LIN {X 0,Y 194.629,Z 450.063,A -85,B 0,C 180,E1 -23083.872,E2 -23083.872} C_VEL
LIN {X 0,Y 195.031,Z 466.842,A -85,B 0,C 180,E1 -23086.302,E2 -23086.302} C_VEL
LIN {X 0,Y 195.009,Z 478.19,A -85,B 0,C 180,E1 -23088.193,E2 -23088.193} C_VEL
LIN {X 0,Y 190.947,Z 492.409,A -85,B 0,C 180,E1 -23090.684,E2 -23090.684} C_VEL
LIN {X 0,Y 187.15,Z 505.053,A -85,B 0,C 180,E1 -23093.413,E2 -23093.413} C_VEL
LIN {X 0,Y 184.446,Z 513.327,A -85,B 0,C 180,E1 -23095.481,E2 -23095.481} C_VEL
LIN {X 0,Y 181.735,Z 524.579,A -85,B 0,C 180,E1 -23097.846,E2 -23097.846} C_VEL
LIN {X 0,Y 179.023,Z 534.861,A -85,B 0,C 180,E1 -23100.619,E2 -23100.619} C_VEL
LIN {X 0,Y 176.653,Z 543.209,A -85,B 0,C 180,E1 -23103.419,E2 -23103.419} C_VEL
LIN {X 0,Y 174.413,Z 551.586,A -85,B 0,C 180,E1 -23106.936,E2 -23106.936} C_VEL
LIN {X 0,Y 173.108,Z 557.098,A -85,B 0,C 180,E1 -23109.819,E2 -23109.819} C_VEL
LIN {X 0,Y 171.926,Z 562.635,A -85,B 0,C 180,E1 -23113.379,E2 -23113.379} C_VEL
LIN {X 0,Y 171.267,Z 566.965,A -85,B 0,C 180,E1 -23116.962,E2 -23116.962} C_VEL
LIN {X 0,Y 171.183,Z 568.089,A -85,B 0,C 180,E1 -23118.106,E2 -23118.106} C_VEL
LIN {X 0,Y 170.832,Z 569.219,A -85,B 0,C 180,E1 -23119.364,E2 -23119.364} C_VEL
LIN {X 0,Y 169.495,Z 570.537,A -85,B 0,C 180,E1 -23121.258,E2 -23121.258} C_VEL
LIN {X 0,Y 165.486,Z 572.266,A -85,B 0,C 180,E1 -23125.813,E2 -23125.813} C_VEL
LIN {X 0,Y 164.692,Z 572.641,A -85,B 0,C 180,E1 -23127.873,E2 -23127.873} C_VEL
LIN {X 0,Y 164.706,Z 572.679,A -85,B 0,C 180,E1 -23128.568,E2 -23128.568} C_VEL
LIN {X 0,Y 164.962,Z 572.852,A -85,B 0,C 180,E1 -23130.006,E2 -23130.006} C_VEL
LIN {X 0,Y 164.703,Z 572.564,A -85,B 0,C 180,E1 -23132.451,E2 -23132.451} C_VEL
LIN {X 0,Y 164.155,Z 571.139,A -85,B 0,C 180,E1 -23137.385,E2 -23137.385} C_VEL
LIN {X 0,Y 163.743,Z 570.715,A -85,B 0,C 180,E1 -23142.398,E2 -23142.398} C_VEL
LIN {X 0,Y 164.326,Z 569.479,A -85,B 0,C 180,E1 -23147.426,E2 -23147.426} C_VEL
LIN {X 0,Y 167.378,Z 566.15,A -85,B 0,C 180,E1 -23154.833,E2 -23154.833} C_VEL
LIN {X 0,Y 173.216,Z 561.282,A -85,B 0,C 180,E1 -23161.84,E2 -23161.84} C_VEL
LIN {X 0,Y 181.825,Z 555.041,A -85,B 0,C 180,E1 -23168.208,E2 -23168.208} C_VEL
LIN {X 0,Y 192.905,Z 547.519,A -85,B 0,C 180,E1 -23173.811,E2 -23173.811} C_VEL
LIN {X 0,Y 203.834,Z 540.338,A -85,B 0,C 180,E1 -23177.848,E2 -23177.848} C_VEL
LIN {X 0,Y 210.94,Z 535.655,A -85,B 0,C 180,E1 -23180.029,E2 -23180.029} C_VEL
LIN {X 0,Y 218.242,Z 530.911,A -85,B 0,C 180,E1 -23181.835,E2 -23181.835} C_VEL
LIN {X 0,Y 219.723,Z 529.675,A -85,B 0,C 180,E1 -23182.575,E2 -23182.575} C_VEL
LIN {X 0,Y 210.166,Z 532.82,A -85,B 0,C 180,E1 -23185.356,E2 -23185.356} C_VEL
LIN {X 0,Y 201.392,Z 535.122,A -85,B 0,C 180,E1 -23188.437,E2 -23188.437} C_VEL
LIN {X 0,Y 193.436,Z 536.513,A -85,B 0,C 180,E1 -23191.816,E2 -23191.816} C_VEL
LIN {X 0,Y 186.362,Z 536.937,A -85,B 0,C 180,E1 -23195.492,E2 -23195.492} C_VEL
LIN {X 0,Y 179.439,Z 536.136,A -85,B 0,C 180,E1 -23200.063,E2 -23200.063} C_VEL
LIN {X 0,Y 175.186,Z 534.57,A -85,B 0,C 180,E1 -23203.692,E2 -23203.692} C_VEL
LIN {X 0,Y 171.279,Z 531.629,A -85,B 0,C 180,E1 -23208.162,E2 -23208.162} C_VEL
LIN {X 0,Y 168.34,Z 527.424,A -85,B 0,C 180,E1 -23212.806,E2 -23212.806} C_VEL
LIN {X 0,Y 166.311,Z 521.843,A -85,B 0,C 180,E1 -23217.579,E2 -23217.579} C_VEL
LIN {X 0,Y 165.364,Z 514.747,A -85,B 0,C 180,E1 -23222.437,E2 -23222.437} C_VEL
LIN {X 0,Y 165.269,Z 507.081,A -85,B 0,C 180,E1 -23226.717,E2 -23226.717} C_VEL
LIN {X 0,Y 165.94,Z 497.974,A -85,B 0,C 180,E1 -23230.988,E2 -23230.988} C_VEL
LIN {X 0,Y 167.032,Z 488.726,A -85,B 0,C 180,E1 -23234.624,E2 -23234.624} C_VEL
LIN {X 0,Y 168.903,Z 476.078,A -85,B 0,C 180,E1 -23238.814,E2 -23238.814} C_VEL
LIN {X 0,Y 170.944,Z 463.074,A -85,B 0,C 180,E1 -23242.353,E2 -23242.353} C_VEL
LIN {X 0,Y 173.422,Z 449.036,A -85,B 0,C 180,E1 -23245.505,E2 -23245.505} C_VEL
LIN {X 0,Y 175.588,Z 435.74,A -85,B 0,C 180,E1 -23248,E2 -23248} C_VEL
LIN {X 0,Y 176.501,Z 428.54,A -85,B 0,C 180,E1 -23249.196,E2 -23249.196} C_VEL
LIN {X 0,Y 174.128,Z 413.815,A -85,B 0,C 180,E1 -23251.784,E2 -23251.784} C_VEL
LIN {X 0,Y 172.139,Z 403.256,A -85,B 0,C 180,E1 -23253.516,E2 -23253.516} C_VEL
LIN {X 0,Y 173.739,Z 403.212,A -85,B 0,C 180,E1 -23254.495,E2 -23254.495} C_VEL
LIN {X 0,Y 176.432,Z 403.928,A -85,B 0,C 180,E1 -23256.693,E2 -23256.693} C_VEL
LIN {X 0,Y 178.16,Z 405.759,A -85,B 0,C 180,E1 -23259.137,E2 -23259.137} C_VEL
LIN {X 0,Y 179.192,Z 408.701,A -85,B 0,C 180,E1 -23261.818,E2 -23261.818} C_VEL
LIN {X 0,Y 179.935,Z 415.092,A -85,B 0,C 180,E1 -23266.573,E2 -23266.573} C_VEL
LIN {X 0,Y 183.206,Z 421.819,A -85,B 0,C 180,E1 -23267.981,E2 -23267.981} C_VEL
LIN {X 0,Y 187.141,Z 432.828,A -85,B 0,C 180,E1 -23270.092,E2 -23270.092} C_VEL
LIN {X 0,Y 189.894,Z 443.18,A -85,B 0,C 180,E1 -23272.163,E2 -23272.163} C_VEL
LIN {X 0,Y 191.456,Z 451.081,A -85,B 0,C 180,E1 -23273.862,E2 -23273.862} C_VEL
LIN {X 0,Y 189.427,Z 461.105,A -85,B 0,C 180,E1 -23275.368,E2 -23275.368} C_VEL
LIN {X 0,Y 186.758,Z 471.226,A -85,B 0,C 180,E1 -23277.246,E2 -23277.246} C_VEL
LIN {X 0,Y 183.655,Z 481.015,A -85,B 0,C 180,E1 -23279.528,E2 -23279.528} C_VEL
LIN {X 0,Y 181.236,Z 488.183,A -85,B 0,C 180,E1 -23281.633,E2 -23281.633} C_VEL
LIN {X 0,Y 177.689,Z 497.048,A -85,B 0,C 180,E1 -23284.832,E2 -23284.832} C_VEL
LIN {X 0,Y 175.128,Z 503.242,A -85,B 0,C 180,E1 -23287.7,E2 -23287.7} C_VEL
LIN {X 0,Y 172.485,Z 508.916,A -85,B 0,C 180,E1 -23290.97,E2 -23290.97} C_VEL
LIN {X 0,Y 170.048,Z 513.577,A -85,B 0,C 180,E1 -23294.411,E2 -23294.411} C_VEL
LIN {X 0,Y 168.231,Z 517.118,A -85,B 0,C 180,E1 -23297.938,E2 -23297.938} C_VEL
LIN {X 0,Y 167.402,Z 518.921,A -85,B 0,C 180,E1 -23300.327,E2 -23300.327} C_VEL
LIN {X 0,Y 166.817,Z 520.285,A -85,B 0,C 180,E1 -23302.733,E2 -23302.733} C_VEL
LIN {X 0,Y 165.996,Z 521.852,A -85,B 0,C 180,E1 -23307.568,E2 -23307.568} C_VEL
LIN {X 0,Y 165.899,Z 522.076,A -85,B 0,C 180,E1 -23309.994,E2 -23309.994} C_VEL
LIN {X 0,Y 166.31,Z 521.305,A -85,B 0,C 180,E1 -23314.842,E2 -23314.842} C_VEL
LIN {X 0,Y 166.835,Z 520.353,A -85,B 0,C 180,E1 -23317.254,E2 -23317.254} C_VEL
LIN {X 0,Y 167.392,Z 519.036,A -85,B 0,C 180,E1 -23319.662,E2 -23319.662} C_VEL
LIN {X 0,Y 168.654,Z 516.249,A -85,B 0,C 180,E1 -23323.243,E2 -23323.243} C_VEL
LIN {X 0,Y 170.716,Z 512.392,A -85,B 0,C 180,E1 -23326.742,E2 -23326.742} C_VEL
LIN {X 0,Y 173.344,Z 507.373,A -85,B 0,C 180,E1 -23330.152,E2 -23330.152} C_VEL
LIN {X 0,Y 176.628,Z 499.912,A -85,B 0,C 180,E1 -23334.063,E2 -23334.063} C_VEL
LIN {X 0,Y 179.855,Z 491.808,A -85,B 0,C 180,E1 -23337.325,E2 -23337.325} C_VEL
LIN {X 0,Y 182.375,Z 485.24,A -85,B 0,C 180,E1 -23339.421,E2 -23339.421} C_VEL
LIN {X 0,Y 185.27,Z 476.452,A -85,B 0,C 180,E1 -23341.751,E2 -23341.751} C_VEL
LIN {X 0,Y 188.331,Z 465.518,A -85,B 0,C 180,E1 -23344.032,E2 -23344.032} C_VEL
LIN {X 0,Y 191.095,Z 454.357,A -85,B 0,C 180,E1 -23345.794,E2 -23345.794} C_VEL
LIN {X 0,Y 191.584,Z 451.553,A -85,B 0,C 180,E1 -23346.191,E2 -23346.191} C_VEL
LIN {X 0,Y 189.429,Z 440.893,A -85,B 0,C 180,E1 -23348.453,E2 -23348.453} C_VEL
LIN {X 0,Y 186.325,Z 429.971,A -85,B 0,C 180,E1 -23350.614,E2 -23350.614} C_VEL
LIN {X 0,Y 182.382,Z 419.877,A -85,B 0,C 180,E1 -23352.58,E2 -23352.58} C_VEL
LIN {X 0,Y 179.899,Z 415.01,A -85,B 0,C 180,E1 -23353.72,E2 -23353.72} C_VEL
LIN {X 0,Y 179.308,Z 408.948,A -85,B 0,C 180,E1 -23358.215,E2 -23358.215} C_VEL
LIN {X 0,Y 178.724,Z 403.336,A -85,B 0,C 180,E1 -23362.777,E2 -23362.777} C_VEL
LIN {X 0,Y 177.867,Z 397.93,A -85,B 0,C 180,E1 -23367.762,E2 -23367.762} C_VEL
LIN {X 0,Y 177.286,Z 394.243,A -85,B 0,C 180,E1 -23371.594,E2 -23371.594} C_VEL
LIN {X 0,Y 176.815,Z 391.984,A -85,B 0,C 180,E1 -23374.072,E2 -23374.072} C_VEL
LIN {X 0,Y 176.477,Z 390.077,A -85,B 0,C 180,E1 -23376.531,E2 -23376.531} C_VEL
LIN {X 0,Y 175.437,Z 386.502,A -85,B 0,C 180,E1 -23381.307,E2 -23381.307} C_VEL
LIN {X 0,Y 174.914,Z 383.609,A -85,B 0,C 180,E1 -23386.049,E2 -23386.049} C_VEL
LIN {X 0,Y 174.725,Z 381.534,A -85,B 0,C 180,E1 -23390.74,E2 -23390.74} C_VEL
LIN {X 0,Y 174.665,Z 380.725,A -85,B 0,C 180,E1 -23393.066,E2 -23393.066} C_VEL
LIN {X 0,Y 174.469,Z 378.781,A -85,B 0,C 180,E1 -23399.999,E2 -23399.999} C_VEL
LIN {X 0,Y 174.677,Z 378.815,A -85,B 0,C 180,E1 -23402.305,E2 -23402.305} C_VEL
LIN {X 0,Y 174.438,Z 379.244,A -85,B 0,C 180,E1 -23404.621,E2 -23404.621} C_VEL
LIN {X 0,Y 173.944,Z 381.469,A -85,B 0,C 180,E1 -23409.3,E2 -23409.3} C_VEL
LIN {X 0,Y 173.968,Z 386.765,A -85,B 0,C 180,E1 -23416.426,E2 -23416.426} C_VEL
LIN {X 0,Y 174.709,Z 390.636,A -85,B 0,C 180,E1 -23420.296,E2 -23420.296} C_VEL
LIN {X 0,Y 175.901,Z 396.13,A -85,B 0,C 180,E1 -23424.803,E2 -23424.803} C_VEL
LIN {X 0,Y 177.591,Z 402.405,A -85,B 0,C 180,E1 -23429.004,E2 -23429.004} C_VEL
LIN {X 0,Y 180.294,Z 412.428,A -85,B 0,C 180,E1 -23434.418,E2 -23434.418} C_VEL
LIN {X 0,Y 182.36,Z 418.529,A -85,B 0,C 180,E1 -23437.371,E2 -23437.371} C_VEL
LIN {X 0,Y 183.06,Z 423.647,A -85,B 0,C 180,E1 -23439.3,E2 -23439.3} C_VEL
LIN {X 0,Y 183.327,Z 425.014,A -85,B 0,C 180,E1 -23439.688,E2 -23439.688} C_VEL
LIN {X 0,Y 187.529,Z 436.693,A -85,B 0,C 180,E1 -23441.459,E2 -23441.459} C_VEL
LIN {X 0,Y 187.863,Z 453.061,A -85,B 0,C 180,E1 -23443.573,E2 -23443.573} C_VEL
LIN {X 0,Y 188.155,Z 468.615,A -85,B 0,C 180,E1 -23445.999,E2 -23445.999} C_VEL
LIN {X 0,Y 188.016,Z 478.475,A -85,B 0,C 180,E1 -23447.722,E2 -23447.722} C_VEL
LIN {X 0,Y 183.619,Z 493.361,A -85,B 0,C 180,E1 -23450.49,E2 -23450.49} C_VEL
LIN {X 0,Y 180.729,Z 502.895,A -85,B 0,C 180,E1 -23452.591,E2 -23452.591} C_VEL
LIN {X 0,Y 178.488,Z 512.207,A -85,B 0,C 180,E1 -23454.155,E2 -23454.155} C_VEL
LIN {X 0,Y 175.885,Z 522.569,A -85,B 0,C 180,E1 -23456.369,E2 -23456.369} C_VEL
LIN {X 0,Y 173.246,Z 531.916,A -85,B 0,C 180,E1 -23458.861,E2 -23458.861} C_VEL
LIN {X 0,Y 170.654,Z 540.567,A -85,B 0,C 180,E1 -23461.739,E2 -23461.739} C_VEL
LIN {X 0,Y 168.108,Z 549.066,A -85,B 0,C 180,E1 -23465.295,E2 -23465.295} C_VEL
LIN {X 0,Y 166.232,Z 556.252,A -85,B 0,C 180,E1 -23469.109,E2 -23469.109} C_VEL
LIN {X 0,Y 165.012,Z 561.529,A -85,B 0,C 180,E1 -23472.661,E2 -23472.661} C_VEL
LIN {X 0,Y 164.278,Z 565.864,A -85,B 0,C 180,E1 -23476.397,E2 -23476.397} C_VEL
LIN {X 0,Y 164.104,Z 569.12,A -85,B 0,C 180,E1 -23480.143,E2 -23480.143} C_VEL
LIN {X 0,Y 164.191,Z 570.709,A -85,B 0,C 180,E1 -23482.628,E2 -23482.628} C_VEL
LIN {X 0,Y 164.314,Z 571.84,A -85,B 0,C 180,E1 -23485.099,E2 -23485.099} C_VEL
LIN {X 0,Y 164.706,Z 572.679,A -85,B 0,C 180,E1 -23488.568,E2 -23488.568} C_VEL
LIN {X 0,Y 164.522,Z 572.784,A -85,B 0,C 180,E1 -23489.925,E2 -23489.925} C_VEL
LIN {X 0,Y 163.204,Z 572.442,A -85,B 0,C 180,E1 -23491.929,E2 -23491.929} C_VEL
LIN {X 0,Y 159.776,Z 571.055,A -85,B 0,C 180,E1 -23495.237,E2 -23495.237} C_VEL
LIN {X 0,Y 157.294,Z 569.602,A -85,B 0,C 180,E1 -23498.384,E2 -23498.384} C_VEL
LIN {X 0,Y 156.984,Z 569.425,A -85,B 0,C 180,E1 -23499.485,E2 -23499.485} C_VEL
LIN {X 0,Y 157.003,Z 568.708,A -85,B 0,C 180,E1 -23505.586,E2 -23505.586} C_VEL
LIN {X 0,Y 159.416,Z 566.2,A -85,B 0,C 180,E1 -23513.383,E2 -23513.383} C_VEL
LIN {X 0,Y 164.677,Z 562.143,A -85,B 0,C 180,E1 -23520.812,E2 -23520.812} C_VEL
LIN {X 0,Y 172.848,Z 556.741,A -85,B 0,C 180,E1 -23527.588,E2 -23527.588} C_VEL
LIN {X 0,Y 183.703,Z 550.114,A -85,B 0,C 180,E1 -23533.528,E2 -23533.528} C_VEL
LIN {X 0,Y 196.757,Z 542.347,A -85,B 0,C 180,E1 -23538.605,E2 -23538.605} C_VEL
LIN {X 0,Y 208.556,Z 535.324,A -85,B 0,C 180,E1 -23542.021,E2 -23542.021} C_VEL
LIN {X 0,Y 209.603,Z 534.353,A -85,B 0,C 180,E1 -23542.877,E2 -23542.877} C_VEL
LIN {X 0,Y 200.13,Z 536.711,A -85,B 0,C 180,E1 -23545.815,E2 -23545.815} C_VEL
LIN {X 0,Y 191.473,Z 538.156,A -85,B 0,C 180,E1 -23549.079,E2 -23549.079} C_VEL
LIN {X 0,Y 183.672,Z 538.688,A -85,B 0,C 180,E1 -23552.668,E2 -23552.668} C_VEL
LIN {X 0,Y 176.77,Z 538.265,A -85,B 0,C 180,E1 -23556.574,E2 -23556.574} C_VEL
LIN {X 0,Y 170.96,Z 536.777,A -85,B 0,C 180,E1 -23560.801,E2 -23560.801} C_VEL
LIN {X 0,Y 166.296,Z 534.137,A -85,B 0,C 180,E1 -23565.312,E2 -23565.312} C_VEL
LIN {X 0,Y 162.654,Z 530.278,A -85,B 0,C 180,E1 -23570.048,E2 -23570.048} C_VEL
LIN {X 0,Y 160.056,Z 525.082,A -85,B 0,C 180,E1 -23574.963,E2 -23574.963} C_VEL
LIN {X 0,Y 158.633,Z 518.447,A -85,B 0,C 180,E1 -23580.001,E2 -23580.001} C_VEL
LIN {X 0,Y 158.181,Z 510.226,A -85,B 0,C 180,E1 -23585.099,E2 -23585.099} C_VEL
LIN {X 0,Y 158.457,Z 501.458,A -85,B 0,C 180,E1 -23589.575,E2 -23589.575} C_VEL
LIN {X 0,Y 159.608,Z 492.066,A -85,B 0,C 180,E1 -23593.628,E2 -23593.628} C_VEL
LIN {X 0,Y 161.17,Z 480.543,A -85,B 0,C 180,E1 -23597.774,E2 -23597.774} C_VEL
LIN {X 0,Y 163.389,Z 467.149,A -85,B 0,C 180,E1 -23601.778,E2 -23601.778} C_VEL
LIN {X 0,Y 165.756,Z 453.791,A -85,B 0,C 180,E1 -23605.088,E2 -23605.088} C_VEL
LIN {X 0,Y 168.612,Z 437.264,A -85,B 0,C 180,E1 -23608.404,E2 -23608.404} C_VEL
LIN {X 0,Y 169.579,Z 429.1,A -85,B 0,C 180,E1 -23609.824,E2 -23609.824} C_VEL
LIN {X 0,Y 167.064,Z 413.363,A -85,B 0,C 180,E1 -23612.708,E2 -23612.708} C_VEL
LIN {X 0,Y 166.063,Z 407.981,A -85,B 0,C 180,E1 -23613.653,E2 -23613.653} C_VEL
LIN {X 0,Y 169.126,Z 407.884,A -85,B 0,C 180,E1 -23615.576,E2 -23615.576} C_VEL
LIN {X 0,Y 171.545,Z 408.948,A -85,B 0,C 180,E1 -23617.919,E2 -23617.919} C_VEL
LIN {X 0,Y 172.4,Z 409.978,A -85,B 0,C 180,E1 -23619.229,E2 -23619.229} C_VEL
LIN {X 0,Y 172.954,Z 411.283,A -85,B 0,C 180,E1 -23620.555,E2 -23620.555} C_VEL
LIN {X 0,Y 173.629,Z 416.288,A -85,B 0,C 180,E1 -23624.553,E2 -23624.553} C_VEL
LIN {X 0,Y 177.596,Z 423.522,A -85,B 0,C 180,E1 -23626.373,E2 -23626.373} C_VEL
LIN {X 0,Y 181.278,Z 433.813,A -85,B 0,C 180,E1 -23628.506,E2 -23628.506} C_VEL
LIN {X 0,Y 183.968,Z 444.245,A -85,B 0,C 180,E1 -23630.705,E2 -23630.705} C_VEL
LIN {X 0,Y 185.658,Z 453.101,A -85,B 0,C 180,E1 -23632.717,E2 -23632.717} C_VEL
LIN {X 0,Y 183.163,Z 464.213,A -85,B 0,C 180,E1 -23634.463,E2 -23634.463} C_VEL
LIN {X 0,Y 179.794,Z 475.77,A -85,B 0,C 180,E1 -23636.816,E2 -23636.816} C_VEL
LIN {X 0,Y 177.05,Z 483.95,A -85,B 0,C 180,E1 -23638.928,E2 -23638.928} C_VEL
LIN {X 0,Y 173.801,Z 492.434,A -85,B 0,C 180,E1 -23641.626,E2 -23641.626} C_VEL
LIN {X 0,Y 170.331,Z 500.662,A -85,B 0,C 180,E1 -23644.975,E2 -23644.975} C_VEL
LIN {X 0,Y 166.808,Z 508.185,A -85,B 0,C 180,E1 -23649.009,E2 -23649.009} C_VEL
LIN {X 0,Y 164.037,Z 513.257,A -85,B 0,C 180,E1 -23652.542,E2 -23652.542} C_VEL
LIN {X 0,Y 161.856,Z 517.167,A -85,B 0,C 180,E1 -23656.177,E2 -23656.177} C_VEL
LIN {X 0,Y 160.486,Z 519.999,A -85,B 0,C 180,E1 -23659.906,E2 -23659.906} C_VEL
LIN {X 0,Y 159.874,Z 521.359,A -85,B 0,C 180,E1 -23662.416,E2 -23662.416} C_VEL
LIN {X 0,Y 158.998,Z 522.927,A -85,B 0,C 180,E1 -23667.46,E2 -23667.46} C_VEL
LIN {X 0,Y 158.909,Z 523.149,A -85,B 0,C 180,E1 -23669.994,E2 -23669.994} C_VEL
LIN {X 0,Y 159.322,Z 522.381,A -85,B 0,C 180,E1 -23675.055,E2 -23675.055} C_VEL
LIN {X 0,Y 159.888,Z 521.428,A -85,B 0,C 180,E1 -23677.571,E2 -23677.571} C_VEL
LIN {X 0,Y 160.475,Z 520.112,A -85,B 0,C 180,E1 -23680.083,E2 -23680.083} C_VEL
LIN {X 0,Y 161.828,Z 517.324,A -85,B 0,C 180,E1 -23683.813,E2 -23683.813} C_VEL
LIN {X 0,Y 164.008,Z 513.466,A -85,B 0,C 180,E1 -23687.449,E2 -23687.449} C_VEL
LIN {X 0,Y 166.774,Z 508.446,A -85,B 0,C 180,E1 -23690.983,E2 -23690.983} C_VEL
LIN {X 0,Y 170.259,Z 500.98,A -85,B 0,C 180,E1 -23695.024,E2 -23695.024} C_VEL
LIN {X 0,Y 173.65,Z 492.876,A -85,B 0,C 180,E1 -23698.388,E2 -23698.388} C_VEL
LIN {X 0,Y 176.293,Z 486.308,A -85,B 0,C 180,E1 -23700.542,E2 -23700.542} C_VEL
LIN {X 0,Y 179.338,Z 477.515,A -85,B 0,C 180,E1 -23702.931,E2 -23702.931} C_VEL
LIN {X 0,Y 182.555,Z 466.574,A -85,B 0,C 180,E1 -23705.265,E2 -23705.265} C_VEL
LIN {X 0,Y 185.411,Z 455.582,A -85,B 0,C 180,E1 -23707.036,E2 -23707.036} C_VEL
LIN {X 0,Y 185.747,Z 453.365,A -85,B 0,C 180,E1 -23707.384,E2 -23707.384} C_VEL
LIN {X 0,Y 183.931,Z 443.684,A -85,B 0,C 180,E1 -23709.567,E2 -23709.567} C_VEL
LIN {X 0,Y 181.13,Z 433.051,A -85,B 0,C 180,E1 -23711.806,E2 -23711.806} C_VEL
LIN {X 0,Y 177.529,Z 423.291,A -85,B 0,C 180,E1 -23713.854,E2 -23713.854} C_VEL
LIN {X 0,Y 173.624,Z 416.324,A -85,B 0,C 180,E1 -23715.651,E2 -23715.651} C_VEL
LIN {X 0,Y 173.12,Z 410.255,A -85,B 0,C 180,E1 -23720.463,E2 -23720.463} C_VEL
LIN {X 0,Y 172.49,Z 404.83,A -85,B 0,C 180,E1 -23725.219,E2 -23725.219} C_VEL
LIN {X 0,Y 171.8,Z 399.531,A -85,B 0,C 180,E1 -23730.599,E2 -23730.599} C_VEL
LIN {X 0,Y 171.522,Z 397.293,A -85,B 0,C 180,E1 -23733.209,E2 -23733.209} C_VEL
LIN {X 0,Y 170.621,Z 393.376,A -85,B 0,C 180,E1 -23738.239,E2 -23738.239} C_VEL
LIN {X 0,Y 169.914,Z 390.111,A -85,B 0,C 180,E1 -23743.169,E2 -23743.169} C_VEL
LIN {X 0,Y 169.817,Z 388.796,A -85,B 0,C 180,E1 -23745.621,E2 -23745.621} C_VEL
LIN {X 0,Y 169.474,Z 386.477,A -85,B 0,C 180,E1 -23750.451,E2 -23750.451} C_VEL
LIN {X 0,Y 169.446,Z 385.416,A -85,B 0,C 180,E1 -23754.446,E2 -23754.446} C_VEL
LIN {X 0,Y 169.662,Z 384.014,A -85,B 0,C 180,E1 -23759.999,E2 -23759.999} C_VEL
LIN {X 0,Y 169.87,Z 384.067,A -85,B 0,C 180,E1 -23762.37,E2 -23762.37} C_VEL
LIN {X 0,Y 169.563,Z 385.221,A -85,B 0,C 180,E1 -23765.945,E2 -23765.945} C_VEL
LIN {X 0,Y 169.203,Z 387.145,A -85,B 0,C 180,E1 -23769.563,E2 -23769.563} C_VEL
LIN {X 0,Y 169.487,Z 392.768,A -85,B 0,C 180,E1 -23776.873,E2 -23776.873} C_VEL
LIN {X 0,Y 170.16,Z 396.597,A -85,B 0,C 180,E1 -23780.552,E2 -23780.552} C_VEL
LIN {X 0,Y 171.629,Z 403.159,A -85,B 0,C 180,E1 -23785.743,E2 -23785.743} C_VEL
LIN {X 0,Y 172.938,Z 408.459,A -85,B 0,C 180,E1 -23789.186,E2 -23789.186} C_VEL
LIN {X 0,Y 176.592,Z 421.301,A -85,B 0,C 180,E1 -23796.072,E2 -23796.072} C_VEL
LIN {X 0,Y 177.328,Z 424.862,A -85,B 0,C 180,E1 -23797.576,E2 -23797.576} C_VEL
LIN {X 0,Y 177.972,Z 430.326,A -85,B 0,C 180,E1 -23799.549,E2 -23799.549} C_VEL
LIN {X 0,Y 180.905,Z 439.096,A -85,B 0,C 180,E1 -23800.944,E2 -23800.944} C_VEL
LIN {X 0,Y 181.071,Z 455.076,A -85,B 0,C 180,E1 -23803.166,E2 -23803.166} C_VEL
LIN {X 0,Y 181.291,Z 471.682,A -85,B 0,C 180,E1 -23805.952,E2 -23805.952} C_VEL
LIN {X 0,Y 181.058,Z 478.546,A -85,B 0,C 180,E1 -23807.222,E2 -23807.222} C_VEL
LIN {X 0,Y 176.937,Z 492.322,A -85,B 0,C 180,E1 -23809.811,E2 -23809.811} C_VEL
LIN {X 0,Y 175.013,Z 501.808,A -85,B 0,C 180,E1 -23811.146,E2 -23811.146} C_VEL
LIN {X 0,Y 172.301,Z 512.55,A -85,B 0,C 180,E1 -23813.021,E2 -23813.021} C_VEL
LIN {X 0,Y 169.258,Z 523.602,A -85,B 0,C 180,E1 -23815.555,E2 -23815.555} C_VEL
LIN {X 0,Y 166.486,Z 532.647,A -85,B 0,C 180,E1 -23818.159,E2 -23818.159} C_VEL
LIN {X 0,Y 163.778,Z 540.993,A -85,B 0,C 180,E1 -23821.142,E2 -23821.142} C_VEL
LIN {X 0,Y 161.142,Z 549.237,A -85,B 0,C 180,E1 -23824.842,E2 -23824.842} C_VEL
LIN {X 0,Y 159.389,Z 555.448,A -85,B 0,C 180,E1 -23828.369,E2 -23828.369} C_VEL
LIN {X 0,Y 158.127,Z 560.422,A -85,B 0,C 180,E1 -23831.88,E2 -23831.88} C_VEL
LIN {X 0,Y 157.285,Z 564.76,A -85,B 0,C 180,E1 -23835.78,E2 -23835.78} C_VEL
LIN {X 0,Y 157.04,Z 568.176,A -85,B 0,C 180,E1 -23839.915,E2 -23839.915} C_VEL
LIN {X 0,Y 157.118,Z 569.615,A -85,B 0,C 180,E1 -23842.295,E2 -23842.295} C_VEL
LIN {X 0,Y 157.256,Z 570.753,A -85,B 0,C 180,E1 -23844.878,E2 -23844.878} C_VEL
LIN {X 0,Y 157.697,Z 571.624,A -85,B 0,C 180,E1 -23848.726,E2 -23848.726} C_VEL
LIN {X 0,Y 157.943,Z 571.775,A -85,B 0,C 180,E1 -23850.006,E2 -23850.006} C_VEL
LIN {X 0,Y 157.648,Z 571.48,A -85,B 0,C 180,E1 -23852.561,E2 -23852.561} C_VEL
LIN {X 0,Y 157.375,Z 570.75,A -85,B 0,C 180,E1 -23855.13,E2 -23855.13} C_VEL
LIN {X 0,Y 157.099,Z 569.46,A -85,B 0,C 180,E1 -23858.409,E2 -23858.409} C_VEL
LIN {X 0,Y 156.984,Z 569.425,A -85,B 0,C 180,E1 -23859.485,E2 -23859.485} C_VEL
LIN {X 0,Y 156.175,Z 569.162,A -85,B 0,C 180,E1 -23861.622,E2 -23861.622} C_VEL
LIN {X 0,Y 153.474,Z 568.078,A -85,B 0,C 180,E1 -23865.132,E2 -23865.132} C_VEL
LIN {X 0,Y 151.562,Z 567.022,A -85,B 0,C 180,E1 -23868.012,E2 -23868.012} C_VEL
LIN {X 0,Y 151.151,Z 566.251,A -85,B 0,C 180,E1 -23870.235,E2 -23870.235} C_VEL
LIN {X 0,Y 151.326,Z 566.025,A -85,B 0,C 180,E1 -23870.977,E2 -23870.977} C_VEL
LIN {X 0,Y 154.358,Z 563.818,A -85,B 0,C 180,E1 -23877.091,E2 -23877.091} C_VEL
LIN {X 0,Y 161.088,Z 559.638,A -85,B 0,C 180,E1 -23884.56,E2 -23884.56} C_VEL
LIN {X 0,Y 170.719,Z 554.225,A -85,B 0,C 180,E1 -23891.205,E2 -23891.205} C_VEL
LIN {X 0,Y 182.85,Z 547.686,A -85,B 0,C 180,E1 -23896.916,E2 -23896.916} C_VEL
LIN {X 0,Y 194.604,Z 541.425,A -85,B 0,C 180,E1 -23900.944,E2 -23900.944} C_VEL
LIN {X 0,Y 200.215,Z 538.395,A -85,B 0,C 180,E1 -23902.547,E2 -23902.547} C_VEL
LIN {X 0,Y 199.408,Z 538.331,A -85,B 0,C 180,E1 -23903.192,E2 -23903.192} C_VEL
LIN {X 0,Y 190.06,Z 539.823,A -85,B 0,C 180,E1 -23906.313,E2 -23906.313} C_VEL
LIN {X 0,Y 181.526,Z 540.485,A -85,B 0,C 180,E1 -23909.782,E2 -23909.782} C_VEL
LIN {X 0,Y 173.871,Z 540.228,A -85,B 0,C 180,E1 -23913.601,E2 -23913.601} C_VEL
LIN {X 0,Y 167.248,Z 538.923,A -85,B 0,C 180,E1 -23917.779,E2 -23917.779} C_VEL
LIN {X 0,Y 161.769,Z 536.526,A -85,B 0,C 180,E1 -23922.296,E2 -23922.296} C_VEL
LIN {X 0,Y 157.476,Z 532.962,A -85,B 0,C 180,E1 -23927.107,E2 -23927.107} C_VEL
LIN {X 0,Y 154.296,Z 528.16,A -85,B 0,C 180,E1 -23932.147,E2 -23932.147} C_VEL
LIN {X 0,Y 152.116,Z 521.975,A -85,B 0,C 180,E1 -23937.353,E2 -23937.353} C_VEL
LIN {X 0,Y 151.148,Z 514.281,A -85,B 0,C 180,E1 -23942.666,E2 -23942.666} C_VEL
LIN {X 0,Y 151.136,Z 506.104,A -85,B 0,C 180,E1 -23947.348,E2 -23947.348} C_VEL
LIN {X 0,Y 151.871,Z 497.389,A -85,B 0,C 180,E1 -23951.561,E2 -23951.561} C_VEL
LIN {X 0,Y 153.095,Z 487.599,A -85,B 0,C 180,E1 -23955.589,E2 -23955.589} C_VEL
LIN {X 0,Y 155.057,Z 475.209,A -85,B 0,C 180,E1 -23959.874,E2 -23959.874} C_VEL
LIN {X 0,Y 157.303,Z 461.795,A -85,B 0,C 180,E1 -23963.711,E2 -23963.711} C_VEL
LIN {X 0,Y 159.986,Z 447.268,A -85,B 0,C 180,E1 -23967.115,E2 -23967.115} C_VEL
LIN {X 0,Y 162.079,Z 435.381,A -85,B 0,C 180,E1 -23969.46,E2 -23969.46} C_VEL
LIN {X 0,Y 162.768,Z 430.867,A -85,B 0,C 180,E1 -23970.272,E2 -23970.272} C_VEL
LIN {X 0,Y 160.74,Z 417.055,A -85,B 0,C 180,E1 -23972.933,E2 -23972.933} C_VEL
LIN {X 0,Y 160.004,Z 412.807,A -85,B 0,C 180,E1 -23973.732,E2 -23973.732} C_VEL
LIN {X 0,Y 164.507,Z 412.689,A -85,B 0,C 180,E1 -23976.735,E2 -23976.735} C_VEL
LIN {X 0,Y 166.63,Z 414.131,A -85,B 0,C 180,E1 -23979.248,E2 -23979.248} C_VEL
LIN {X 0,Y 167.387,Z 417.487,A -85,B 0,C 180,E1 -23982.296,E2 -23982.296} C_VEL
LIN {X 0,Y 172.936,Z 427.367,A -85,B 0,C 180,E1 -23985.126,E2 -23985.126} C_VEL
LIN {X 0,Y 176.221,Z 437.232,A -85,B 0,C 180,E1 -23987.336,E2 -23987.336} C_VEL
LIN {X 0,Y 178.551,Z 447.231,A -85,B 0,C 180,E1 -23989.596,E2 -23989.596} C_VEL
LIN {X 0,Y 179.863,Z 454.72,A -85,B 0,C 180,E1 -23991.398,E2 -23991.398} C_VEL
LIN {X 0,Y 179.855,Z 456.025,A -85,B 0,C 180,E1 -23991.665,E2 -23991.665} C_VEL
LIN {X 0,Y 176.981,Z 466.896,A -85,B 0,C 180,E1 -23993.435,E2 -23993.435} C_VEL
LIN {X 0,Y 173.578,Z 477.97,A -85,B 0,C 180,E1 -23995.815,E2 -23995.815} C_VEL
LIN {X 0,Y 171.076,Z 485.022,A -85,B 0,C 180,E1 -23997.714,E2 -23997.714} C_VEL
LIN {X 0,Y 167.683,Z 493.503,A -85,B 0,C 180,E1 -24000.491,E2 -24000.491} C_VEL
LIN {X 0,Y 164.02,Z 501.734,A -85,B 0,C 180,E1 -24003.941,E2 -24003.941} C_VEL
LIN {X 0,Y 161.327,Z 507.316,A -85,B 0,C 180,E1 -24006.91,E2 -24006.91} C_VEL
LIN {X 0,Y 158.363,Z 512.76,A -85,B 0,C 180,E1 -24010.553,E2 -24010.553} C_VEL
LIN {X 0,Y 155.687,Z 517.061,A -85,B 0,C 180,E1 -24014.279,E2 -24014.279} C_VEL
LIN {X 0,Y 154.527,Z 519.274,A -85,B 0,C 180,E1 -24016.85,E2 -24016.85} C_VEL
LIN {X 0,Y 153.579,Z 521.077,A -85,B 0,C 180,E1 -24019.447,E2 -24019.447} C_VEL
LIN {X 0,Y 152.933,Z 522.435,A -85,B 0,C 180,E1 -24022.069,E2 -24022.069} C_VEL
LIN {X 0,Y 151.998,Z 524.002,A -85,B 0,C 180,E1 -24027.343,E2 -24027.343} C_VEL
LIN {X 0,Y 151.915,Z 524.223,A -85,B 0,C 180,E1 -24029.994,E2 -24029.994} C_VEL
LIN {X 0,Y 152.335,Z 523.457,A -85,B 0,C 180,E1 -24035.288,E2 -24035.288} C_VEL
LIN {X 0,Y 152.943,Z 522.502,A -85,B 0,C 180,E1 -24037.917,E2 -24037.917} C_VEL
LIN {X 0,Y 153.567,Z 521.189,A -85,B 0,C 180,E1 -24040.541,E2 -24040.541} C_VEL
LIN {X 0,Y 155.02,Z 518.4,A -85,B 0,C 180,E1 -24044.432,E2 -24044.432} C_VEL
LIN {X 0,Y 157.328,Z 514.54,A -85,B 0,C 180,E1 -24048.215,E2 -24048.215} C_VEL
LIN {X 0,Y 160.243,Z 509.518,A -85,B 0,C 180,E1 -24051.881,E2 -24051.881} C_VEL
LIN {X 0,Y 163.946,Z 502.049,A -85,B 0,C 180,E1 -24056.058,E2 -24056.058} C_VEL
LIN {X 0,Y 167.509,Z 493.945,A -85,B 0,C 180,E1 -24059.529,E2 -24059.529} C_VEL
LIN {X 0,Y 170.283,Z 487.375,A -85,B 0,C 180,E1 -24061.743,E2 -24061.743} C_VEL
LIN {X 0,Y 173.488,Z 478.578,A -85,B 0,C 180,E1 -24064.192,E2 -24064.192} C_VEL
LIN {X 0,Y 176.87,Z 467.632,A -85,B 0,C 180,E1 -24066.578,E2 -24066.578} C_VEL
LIN {X 0,Y 179.866,Z 456.634,A -85,B 0,C 180,E1 -24068.379,E2 -24068.379} C_VEL
LIN {X 0,Y 179.842,Z 454.229,A -85,B 0,C 180,E1 -24068.886,E2 -24068.886} C_VEL
LIN {X 0,Y 177.906,Z 443.773,A -85,B 0,C 180,E1 -24071.358,E2 -24071.358} C_VEL
LIN {X 0,Y 175.489,Z 434.395,A -85,B 0,C 180,E1 -24073.447,E2 -24073.447} C_VEL
LIN {X 0,Y 172.804,Z 427.143,A -85,B 0,C 180,E1 -24075.139,E2 -24075.139} C_VEL
LIN {X 0,Y 168.941,Z 420.338,A -85,B 0,C 180,E1 -24077.068,E2 -24077.068} C_VEL
LIN {X 0,Y 167.456,Z 417.518,A -85,B 0,C 180,E1 -24077.898,E2 -24077.898} C_VEL
LIN {X 0,Y 167.03,Z 412.159,A -85,B 0,C 180,E1 -24082.403,E2 -24082.403} C_VEL
LIN {X 0,Y 166.546,Z 407.625,A -85,B 0,C 180,E1 -24086.729,E2 -24086.729} C_VEL
LIN {X 0,Y 166.145,Z 403.716,A -85,B 0,C 180,E1 -24090.891,E2 -24090.891} C_VEL
LIN {X 0,Y 165.708,Z 400.504,A -85,B 0,C 180,E1 -24094.904,E2 -24094.904} C_VEL
LIN {X 0,Y 164.895,Z 396.779,A -85,B 0,C 180,E1 -24100.063,E2 -24100.063} C_VEL
LIN {X 0,Y 164.544,Z 393.864,A -85,B 0,C 180,E1 -24105.15,E2 -24105.15} C_VEL
LIN {X 0,Y 164.523,Z 391.723,A -85,B 0,C 180,E1 -24110.161,E2 -24110.161} C_VEL
LIN {X 0,Y 164.431,Z 390.801,A -85,B 0,C 180,E1 -24112.632,E2 -24112.632} C_VEL
LIN {X 0,Y 164.853,Z 389.249,A -85,B 0,C 180,E1 -24119.999,E2 -24119.999} C_VEL
LIN {X 0,Y 165.051,Z 389.318,A -85,B 0,C 180,E1 -24122.439,E2 -24122.439} C_VEL
LIN {X 0,Y 164.909,Z 390.084,A -85,B 0,C 180,E1 -24124.889,E2 -24124.889} C_VEL
LIN {X 0,Y 164.506,Z 392.851,A -85,B 0,C 180,E1 -24129.838,E2 -24129.838} C_VEL
LIN {X 0,Y 164.767,Z 397.676,A -85,B 0,C 180,E1 -24136.095,E2 -24136.095} C_VEL
LIN {X 0,Y 165.437,Z 401.506,A -85,B 0,C 180,E1 -24139.867,E2 -24139.867} C_VEL
LIN {X 0,Y 166.689,Z 407.739,A -85,B 0,C 180,E1 -24144.936,E2 -24144.936} C_VEL
LIN {X 0,Y 168.021,Z 413.222,A -85,B 0,C 180,E1 -24148.566,E2 -24148.566} C_VEL
LIN {X 0,Y 171.092,Z 424.931,A -85,B 0,C 180,E1 -24155.104,E2 -24155.104} C_VEL
LIN {X 0,Y 171.749,Z 427.657,A -85,B 0,C 180,E1 -24156.394,E2 -24156.394} C_VEL
LIN {X 0,Y 172.696,Z 436.095,A -85,B 0,C 180,E1 -24159.567,E2 -24159.567} C_VEL
LIN {X 0,Y 174.209,Z 440.906,A -85,B 0,C 180,E1 -24160.39,E2 -24160.39} C_VEL
LIN {X 0,Y 174.298,Z 457.55,A -85,B 0,C 180,E1 -24162.876,E2 -24162.876} C_VEL
LIN {X 0,Y 174.37,Z 473.67,A -85,B 0,C 180,E1 -24165.762,E2 -24165.762} C_VEL
LIN {X 0,Y 174.128,Z 478.423,A -85,B 0,C 180,E1 -24166.684,E2 -24166.684} C_VEL
LIN {X 0,Y 173.391,Z 480.764,A -85,B 0,C 180,E1 -24167.119,E2 -24167.119} C_VEL
LIN {X 0,Y 171.595,Z 490.581,A -85,B 0,C 180,E1 -24168.169,E2 -24168.169} C_VEL
LIN {X 0,Y 169.055,Z 502.43,A -85,B 0,C 180,E1 -24169.89,E2 -24169.89} C_VEL
LIN {X 0,Y 166.181,Z 512.783,A -85,B 0,C 180,E1 -24171.801,E2 -24171.801} C_VEL
LIN {X 0,Y 162.976,Z 523.589,A -85,B 0,C 180,E1 -24174.406,E2 -24174.406} C_VEL
LIN {X 0,Y 159.66,Z 533.616,A -85,B 0,C 180,E1 -24177.48,E2 -24177.48} C_VEL
LIN {X 0,Y 156.415,Z 542.816,A -85,B 0,C 180,E1 -24181.125,E2 -24181.125} C_VEL
LIN {X 0,Y 153.835,Z 550.487,A -85,B 0,C 180,E1 -24185.01,E2 -24185.01} C_VEL
LIN {X 0,Y 152.242,Z 555.739,A -85,B 0,C 180,E1 -24188.335,E2 -24188.335} C_VEL
LIN {X 0,Y 150.868,Z 560.863,A -85,B 0,C 180,E1 -24192.382,E2 -24192.382} C_VEL
LIN {X 0,Y 150.118,Z 564.834,A -85,B 0,C 180,E1 -24196.47,E2 -24196.47} C_VEL
LIN {X 0,Y 149.992,Z 567.254,A -85,B 0,C 180,E1 -24199.722,E2 -24199.722} C_VEL
LIN {X 0,Y 150.051,Z 568.52,A -85,B 0,C 180,E1 -24201.929,E2 -24201.929} C_VEL
LIN {X 0,Y 150.199,Z 569.666,A -85,B 0,C 180,E1 -24204.637,E2 -24204.637} C_VEL
LIN {X 0,Y 150.47,Z 570.39,A -85,B 0,C 180,E1 -24207.329,E2 -24207.329} C_VEL
LIN {X 0,Y 150.92,Z 570.697,A -85,B 0,C 180,E1 -24210.006,E2 -24210.006} C_VEL
LIN {X 0,Y 150.588,Z 570.395,A -85,B 0,C 180,E1 -24212.681,E2 -24212.681} C_VEL
LIN {X 0,Y 150.3,Z 569.659,A -85,B 0,C 180,E1 -24215.373,E2 -24215.373} C_VEL
LIN {X 0,Y 150.071,Z 567.698,A -85,B 0,C 180,E1 -24219.824,E2 -24219.824} C_VEL
LIN {X 0,Y 150.16,Z 567.099,A -85,B 0,C 180,E1 -24226.316,E2 -24226.316} C_VEL
LIN {X 0,Y 151.326,Z 566.025,A -85,B 0,C 180,E1 -24230.977,E2 -24230.977} C_VEL
LIN {X 0,Y 151.565,Z 565.269,A -85,B 0,C 180,E1 -24233.19,E2 -24233.19} C_VEL
LIN {X 0,Y 150.648,Z 563.568,A -85,B 0,C 180,E1 -24236.879,E2 -24236.879} C_VEL
LIN {X 0,Y 150.249,Z 562.031,A -85,B 0,C 180,E1 -24239.847,E2 -24239.847} C_VEL
LIN {X 0,Y 151.019,Z 560.895,A -85,B 0,C 180,E1 -24242.035,E2 -24242.035} C_VEL
LIN {X 0,Y 151.589,Z 560.53,A -85,B 0,C 180,E1 -24242.736,E2 -24242.736} C_VEL
LIN {X 0,Y 158.28,Z 557.151,A -85,B 0,C 180,E1 -24248.442,E2 -24248.442} C_VEL
LIN {X 0,Y 169.338,Z 551.779,A -85,B 0,C 180,E1 -24254.881,E2 -24254.881} C_VEL
LIN {X 0,Y 182.728,Z 545.387,A -85,B 0,C 180,E1 -24260.292,E2 -24260.292} C_VEL
LIN {X 0,Y 189.292,Z 542.26,A -85,B 0,C 180,E1 -24262.346,E2 -24262.346} C_VEL
LIN {X 0,Y 190.258,Z 541.48,A -85,B 0,C 180,E1 -24263.173,E2 -24263.173} C_VEL
LIN {X 0,Y 179.936,Z 542.305,A -85,B 0,C 180,E1 -24266.852,E2 -24266.852} C_VEL
LIN {X 0,Y 171.535,Z 542.121,A -85,B 0,C 180,E1 -24270.552,E2 -24270.552} C_VEL
LIN {X 0,Y 164.094,Z 541.006,A -85,B 0,C 180,E1 -24274.642,E2 -24274.642} C_VEL
LIN {X 0,Y 157.772,Z 538.856,A -85,B 0,C 180,E1 -24279.124,E2 -24279.124} C_VEL
LIN {X 0,Y 152.692,Z 535.574,A -85,B 0,C 180,E1 -24283.97,E2 -24283.97} C_VEL
LIN {X 0,Y 148.74,Z 531.106,A -85,B 0,C 180,E1 -24289.107,E2 -24289.107} C_VEL
LIN {X 0,Y 145.94,Z 525.322,A -85,B 0,C 180,E1 -24294.474,E2 -24294.474} C_VEL
LIN {X 0,Y 144.4,Z 518.064,A -85,B 0,C 180,E1 -24300.001,E2 -24300.001} C_VEL
LIN {X 0,Y 144.001,Z 510.416,A -85,B 0,C 180,E1 -24304.901,E2 -24304.901} C_VEL
LIN {X 0,Y 144.433,Z 499.863,A -85,B 0,C 180,E1 -24310.515,E2 -24310.515} C_VEL
LIN {X 0,Y 145.441,Z 492.179,A -85,B 0,C 180,E1 -24313.983,E2 -24313.983} C_VEL
LIN {X 0,Y 147.261,Z 479.625,A -85,B 0,C 180,E1 -24318.794,E2 -24318.794} C_VEL
LIN {X 0,Y 149.711,Z 465.796,A -85,B 0,C 180,E1 -24323.152,E2 -24323.152} C_VEL
LIN {X 0,Y 152.353,Z 451.888,A -85,B 0,C 180,E1 -24326.73,E2 -24326.73} C_VEL
LIN {X 0,Y 155.087,Z 436.877,A -85,B 0,C 180,E1 -24329.901,E2 -24329.901} C_VEL
LIN {X 0,Y 155.83,Z 430.979,A -85,B 0,C 180,E1 -24331.019,E2 -24331.019} C_VEL
LIN {X 0,Y 153.867,Z 417.589,A -85,B 0,C 180,E1 -24333.788,E2 -24333.788} C_VEL
LIN {X 0,Y 154.736,Z 417.664,A -85,B 0,C 180,E1 -24334.533,E2 -24334.533} C_VEL
LIN {X 0,Y 159.311,Z 417.32,A -85,B 0,C 180,E1 -24337.424,E2 -24337.424} C_VEL
LIN {X 0,Y 160.877,Z 418.419,A -85,B 0,C 180,E1 -24339.306,E2 -24339.306} C_VEL
LIN {X 0,Y 161.202,Z 419.218,A -85,B 0,C 180,E1 -24339.92,E2 -24339.92} C_VEL
LIN {X 0,Y 164.824,Z 424.846,A -85,B 0,C 180,E1 -24341.867,E2 -24341.867} C_VEL
LIN {X 0,Y 168.662,Z 432.042,A -85,B 0,C 180,E1 -24344.057,E2 -24344.057} C_VEL
LIN {X 0,Y 171.717,Z 442.619,A -85,B 0,C 180,E1 -24346.592,E2 -24346.592} C_VEL
LIN {X 0,Y 173.796,Z 454.015,A -85,B 0,C 180,E1 -24349.388,E2 -24349.388} C_VEL
LIN {X 0,Y 174.264,Z 457.275,A -85,B 0,C 180,E1 -24350.234,E2 -24350.234} C_VEL
LIN {X 0,Y 171.395,Z 467.962,A -85,B 0,C 180,E1 -24352.037,E2 -24352.037} C_VEL
LIN {X 0,Y 167.817,Z 479.04,A -85,B 0,C 180,E1 -24354.468,E2 -24354.468} C_VEL
LIN {X 0,Y 165.183,Z 486.094,A -85,B 0,C 180,E1 -24356.413,E2 -24356.413} C_VEL
LIN {X 0,Y 161.63,Z 494.574,A -85,B 0,C 180,E1 -24359.269,E2 -24359.269} C_VEL
LIN {X 0,Y 158.319,Z 501.564,A -85,B 0,C 180,E1 -24362.212,E2 -24362.212} C_VEL
LIN {X 0,Y 154.901,Z 508.392,A -85,B 0,C 180,E1 -24365.893,E2 -24365.893} C_VEL
LIN {X 0,Y 151.778,Z 513.835,A -85,B 0,C 180,E1 -24369.672,E2 -24369.672} C_VEL
LIN {X 0,Y 148.945,Z 518.138,A -85,B 0,C 180,E1 -24373.548,E2 -24373.548} C_VEL
LIN {X 0,Y 147.698,Z 520.352,A -85,B 0,C 180,E1 -24376.23,E2 -24376.23} C_VEL
LIN {X 0,Y 146.683,Z 522.155,A -85,B 0,C 180,E1 -24378.944,E2 -24378.944} C_VEL
LIN {X 0,Y 145.995,Z 523.51,A -85,B 0,C 180,E1 -24381.69,E2 -24381.69} C_VEL
LIN {X 0,Y 145.015,Z 525.075,A -85,B 0,C 180,E1 -24387.215,E2 -24387.215} C_VEL
LIN {X 0,Y 144.917,Z 525.297,A -85,B 0,C 180,E1 -24389.993,E2 -24389.993} C_VEL
LIN {X 0,Y 145.351,Z 524.533,A -85,B 0,C 180,E1 -24395.543,E2 -24395.543} C_VEL
LIN {X 0,Y 146.002,Z 523.578,A -85,B 0,C 180,E1 -24398.296,E2 -24398.296} C_VEL
LIN {X 0,Y 146.67,Z 522.265,A -85,B 0,C 180,E1 -24401.043,E2 -24401.043} C_VEL
LIN {X 0,Y 148.232,Z 519.475,A -85,B 0,C 180,E1 -24405.108,E2 -24405.108} C_VEL
LIN {X 0,Y 150.678,Z 515.614,A -85,B 0,C 180,E1 -24409.049,E2 -24409.049} C_VEL
LIN {X 0,Y 153.754,Z 510.591,A -85,B 0,C 180,E1 -24412.856,E2 -24412.856} C_VEL
LIN {X 0,Y 157.669,Z 503.12,A -85,B 0,C 180,E1 -24417.179,E2 -24417.179} C_VEL
LIN {X 0,Y 161.439,Z 495.013,A -85,B 0,C 180,E1 -24420.757,E2 -24420.757} C_VEL
LIN {X 0,Y 164.354,Z 488.442,A -85,B 0,C 180,E1 -24423.031,E2 -24423.031} C_VEL
LIN {X 0,Y 167.727,Z 479.641,A -85,B 0,C 180,E1 -24425.54,E2 -24425.54} C_VEL
LIN {X 0,Y 171.284,Z 468.689,A -85,B 0,C 180,E1 -24427.978,E2 -24427.978} C_VEL
LIN {X 0,Y 174.36,Z 457.841,A -85,B 0,C 180,E1 -24429.793,E2 -24429.793} C_VEL
LIN {X 0,Y 172.874,Z 447.851,A -85,B 0,C 180,E1 -24432.317,E2 -24432.317} C_VEL
LIN {X 0,Y 170.5,Z 437.666,A -85,B 0,C 180,E1 -24434.769,E2 -24434.769} C_VEL
LIN {X 0,Y 168.43,Z 431.581,A -85,B 0,C 180,E1 -24436.282,E2 -24436.282} C_VEL
LIN {X 0,Y 163.535,Z 422.531,A -85,B 0,C 180,E1 -24439.066,E2 -24439.066} C_VEL
LIN {X 0,Y 161.365,Z 418.815,A -85,B 0,C 180,E1 -24440.332,E2 -24440.332} C_VEL
LIN {X 0,Y 161.16,Z 414.877,A -85,B 0,C 180,E1 -24443.933,E2 -24443.933} C_VEL
LIN {X 0,Y 160.769,Z 410.57,A -85,B 0,C 180,E1 -24448.359,E2 -24448.359} C_VEL
LIN {X 0,Y 160.423,Z 406.725,A -85,B 0,C 180,E1 -24452.746,E2 -24452.746} C_VEL
LIN {X 0,Y 159.885,Z 403.339,A -85,B 0,C 180,E1 -24457.363,E2 -24457.363} C_VEL
LIN {X 0,Y 159.435,Z 400.43,A -85,B 0,C 180,E1 -24462.026,E2 -24462.026} C_VEL
LIN {X 0,Y 159.388,Z 398.477,A -85,B 0,C 180,E1 -24465.915,E2 -24465.915} C_VEL
LIN {X 0,Y 159.321,Z 396.771,A -85,B 0,C 180,E1 -24469.836,E2 -24469.836} C_VEL
LIN {X 0,Y 159.478,Z 396.022,A -85,B 0,C 180,E1 -24472.402,E2 -24472.402} C_VEL
LIN {X 0,Y 160.066,Z 394.529,A -85,B 0,C 180,E1 -24479.999,E2 -24479.999} C_VEL
LIN {X 0,Y 160.366,Z 394.716,A -85,B 0,C 180,E1 -24482.511,E2 -24482.511} C_VEL
LIN {X 0,Y 160.162,Z 395.586,A -85,B 0,C 180,E1 -24485.034,E2 -24485.034} C_VEL
LIN {X 0,Y 159.894,Z 396.884,A -85,B 0,C 180,E1 -24487.576,E2 -24487.576} C_VEL
LIN {X 0,Y 159.819,Z 400.519,A -85,B 0,C 180,E1 -24492.701,E2 -24492.701} C_VEL
LIN {X 0,Y 160.21,Z 403.677,A -85,B 0,C 180,E1 -24496.566,E2 -24496.566} C_VEL
LIN {X 0,Y 161.128,Z 409.267,A -85,B 0,C 180,E1 -24501.691,E2 -24501.691} C_VEL
LIN {X 0,Y 162.194,Z 414.395,A -85,B 0,C 180,E1 -24505.677,E2 -24505.677} C_VEL
LIN {X 0,Y 163.717,Z 421.599,A -85,B 0,C 180,E1 -24510.194,E2 -24510.194} C_VEL
LIN {X 0,Y 165.944,Z 429.957,A -85,B 0,C 180,E1 -24514.86,E2 -24514.86} C_VEL
LIN {X 0,Y 166.38,Z 434.066,A -85,B 0,C 180,E1 -24516.635,E2 -24516.635} C_VEL
LIN {X 0,Y 167.238,Z 441.594,A -85,B 0,C 180,E1 -24519.638,E2 -24519.638} C_VEL
LIN {X 0,Y 167.507,Z 450.213,A -85,B 0,C 180,E1 -24520.966,E2 -24520.966} C_VEL
LIN {X 0,Y 167.471,Z 465.507,A -85,B 0,C 180,E1 -24523.494,E2 -24523.494} C_VEL
LIN {X 0,Y 168.203,Z 479.341,A -85,B 0,C 180,E1 -24525.399,E2 -24525.399} C_VEL
LIN {X 0,Y 166.024,Z 490.831,A -85,B 0,C 180,E1 -24526.681,E2 -24526.681} C_VEL
LIN {X 0,Y 163.536,Z 501.334,A -85,B 0,C 180,E1 -24528.241,E2 -24528.241} C_VEL
LIN {X 0,Y 160.148,Z 512.997,A -85,B 0,C 180,E1 -24530.491,E2 -24530.491} C_VEL
LIN {X 0,Y 156.762,Z 523.578,A -85,B 0,C 180,E1 -24533.165,E2 -24533.165} C_VEL
LIN {X 0,Y 153.508,Z 532.756,A -85,B 0,C 180,E1 -24536.114,E2 -24536.114} C_VEL
LIN {X 0,Y 150.096,Z 541.708,A -85,B 0,C 180,E1 -24539.786,E2 -24539.786} C_VEL
LIN {X 0,Y 147.254,Z 549.372,A -85,B 0,C 180,E1 -24543.81,E2 -24543.81} C_VEL
LIN {X 0,Y 145.503,Z 554.626,A -85,B 0,C 180,E1 -24547.276,E2 -24547.276} C_VEL
LIN {X 0,Y 144,Z 559.757,A -85,B 0,C 180,E1 -24551.512,E2 -24551.512} C_VEL
LIN {X 0,Y 143.112,Z 563.728,A -85,B 0,C 180,E1 -24555.794,E2 -24555.794} C_VEL
LIN {X 0,Y 142.946,Z 566.328,A -85,B 0,C 180,E1 -24559.511,E2 -24559.511} C_VEL
LIN {X 0,Y 143.141,Z 568.578,A -85,B 0,C 180,E1 -24564.372,E2 -24564.372} C_VEL
LIN {X 0,Y 143.408,Z 569.306,A -85,B 0,C 180,E1 -24567.198,E2 -24567.198} C_VEL
LIN {X 0,Y 143.893,Z 569.619,A -85,B 0,C 180,E1 -24570.007,E2 -24570.007} C_VEL
LIN {X 0,Y 143.524,Z 569.31,A -85,B 0,C 180,E1 -24572.814,E2 -24572.814} C_VEL
LIN {X 0,Y 143.232,Z 568.569,A -85,B 0,C 180,E1 -24575.638,E2 -24575.638} C_VEL
LIN {X 0,Y 143.051,Z 566.177,A -85,B 0,C 180,E1 -24580.714,E2 -24580.714} C_VEL
LIN {X 0,Y 143.066,Z 565.826,A -85,B 0,C 180,E1 -24581.339,E2 -24581.339} C_VEL
LIN {X 0,Y 143.343,Z 565.466,A -85,B 0,C 180,E1 -24587.115,E2 -24587.115} C_VEL
LIN {X 0,Y 146.319,Z 563.494,A -85,B 0,C 180,E1 -24595.62,E2 -24595.62} C_VEL
LIN {X 0,Y 151.589,Z 560.53,A -85,B 0,C 180,E1 -24602.736,E2 -24602.736} C_VEL
LIN {X 0,Y 153.052,Z 559.399,A -85,B 0,C 180,E1 -24604.848,E2 -24604.848} C_VEL
LIN {X 0,Y 156.202,Z 555.024,A -85,B 0,C 180,E1 -24611.917,E2 -24611.917} C_VEL
LIN {X 0,Y 158.665,Z 553.665,A -85,B 0,C 180,E1 -24613.801,E2 -24613.801} C_VEL
LIN {X 0,Y 168.753,Z 549.414,A -85,B 0,C 180,E1 -24618.567,E2 -24618.567} C_VEL
LIN {X 0,Y 178.255,Z 545.353,A -85,B 0,C 180,E1 -24622.056,E2 -24622.056} C_VEL
LIN {X 0,Y 180.341,Z 544.059,A -85,B 0,C 180,E1 -24623.405,E2 -24623.405} C_VEL
LIN {X 0,Y 169.775,Z 544.042,A -85,B 0,C 180,E1 -24627.444,E2 -24627.444} C_VEL
LIN {X 0,Y 161.517,Z 543.1,A -85,B 0,C 180,E1 -24631.405,E2 -24631.405} C_VEL
LIN {X 0,Y 154.363,Z 541.121,A -85,B 0,C 180,E1 -24635.811,E2 -24635.811} C_VEL
LIN {X 0,Y 148.426,Z 538.061,A -85,B 0,C 180,E1 -24640.644,E2 -24640.644} C_VEL
LIN {X 0,Y 143.725,Z 533.868,A -85,B 0,C 180,E1 -24645.849,E2 -24645.849} C_VEL
LIN {X 0,Y 140.245,Z 528.45,A -85,B 0,C 180,E1 -24651.355,E2 -24651.355} C_VEL
LIN {X 0,Y 137.947,Z 521.671,A -85,B 0,C 180,E1 -24657.081,E2 -24657.081} C_VEL
LIN {X 0,Y 136.956,Z 513.334,A -85,B 0,C 180,E1 -24662.943,E2 -24662.943} C_VEL
LIN {X 0,Y 137.037,Z 504.606,A -85,B 0,C 180,E1 -24668.109,E2 -24668.109} C_VEL
LIN {X 0,Y 138.157,Z 494.217,A -85,B 0,C 180,E1 -24673.234,E2 -24673.234} C_VEL
LIN {X 0,Y 139.859,Z 481.937,A -85,B 0,C 180,E1 -24678.306,E2 -24678.306} C_VEL
LIN {X 0,Y 142.016,Z 469.475,A -85,B 0,C 180,E1 -24682.553,E2 -24682.553} C_VEL
LIN {X 0,Y 144.86,Z 454.813,A -85,B 0,C 180,E1 -24686.666,E2 -24686.666} C_VEL
LIN {X 0,Y 147.682,Z 440.386,A -85,B 0,C 180,E1 -24689.98,E2 -24689.98} C_VEL
LIN {X 0,Y 148.974,Z 432.296,A -85,B 0,C 180,E1 -24691.583,E2 -24691.583} C_VEL
LIN {X 0,Y 147.874,Z 423.942,A -85,B 0,C 180,E1 -24693.418,E2 -24693.418} C_VEL
LIN {X 0,Y 148.331,Z 424.564,A -85,B 0,C 180,E1 -24693.749,E2 -24693.749} C_VEL
LIN {X 0,Y 149.717,Z 424.626,A -85,B 0,C 180,E1 -24694.571,E2 -24694.571} C_VEL
LIN {X 0,Y 151.136,Z 423.467,A -85,B 0,C 180,E1 -24695.275,E2 -24695.275} C_VEL
LIN {X 0,Y 156.041,Z 423.657,A -85,B 0,C 180,E1 -24697.852,E2 -24697.852} C_VEL
LIN {X 0,Y 158.039,Z 424.969,A -85,B 0,C 180,E1 -24698.914,E2 -24698.914} C_VEL
LIN {X 0,Y 161.295,Z 430.456,A -85,B 0,C 180,E1 -24700.917,E2 -24700.917} C_VEL
LIN {X 0,Y 164.334,Z 436.755,A -85,B 0,C 180,E1 -24702.97,E2 -24702.97} C_VEL
LIN {X 0,Y 166.658,Z 445.921,A -85,B 0,C 180,E1 -24705.326,E2 -24705.326} C_VEL
LIN {X 0,Y 168.351,Z 456.488,A -85,B 0,C 180,E1 -24708.085,E2 -24708.085} C_VEL
LIN {X 0,Y 168.669,Z 459.504,A -85,B 0,C 180,E1 -24708.909,E2 -24708.909} C_VEL
LIN {X 0,Y 165.532,Z 470.39,A -85,B 0,C 180,E1 -24710.829,E2 -24710.829} C_VEL
LIN {X 0,Y 161.731,Z 481.208,A -85,B 0,C 180,E1 -24713.302,E2 -24713.302} C_VEL
LIN {X 0,Y 158.687,Z 489.023,A -85,B 0,C 180,E1 -24715.613,E2 -24715.613} C_VEL
LIN {X 0,Y 154.917,Z 497.163,A -85,B 0,C 180,E1 -24718.546,E2 -24718.546} C_VEL
LIN {X 0,Y 150.907,Z 505.066,A -85,B 0,C 180,E1 -24722.237,E2 -24722.237} C_VEL
LIN {X 0,Y 147.351,Z 511.413,A -85,B 0,C 180,E1 -24726.076,E2 -24726.076} C_VEL
LIN {X 0,Y 144.094,Z 516.488,A -85,B 0,C 180,E1 -24730.03,E2 -24730.03} C_VEL
LIN {X 0,Y 141.497,Z 520.4,A -85,B 0,C 180,E1 -24734.14,E2 -24734.14} C_VEL
LIN {X 0,Y 139.8,Z 523.232,A -85,B 0,C 180,E1 -24738.393,E2 -24738.393} C_VEL
LIN {X 0,Y 139.061,Z 524.587,A -85,B 0,C 180,E1 -24741.272,E2 -24741.272} C_VEL
LIN {X 0,Y 138.029,Z 526.149,A -85,B 0,C 180,E1 -24747.074,E2 -24747.074} C_VEL
LIN {X 0,Y 137.916,Z 526.371,A -85,B 0,C 180,E1 -24749.993,E2 -24749.993} C_VEL
LIN {X 0,Y 138.368,Z 525.61,A -85,B 0,C 180,E1 -24755.823,E2 -24755.823} C_VEL
LIN {X 0,Y 139.066,Z 524.653,A -85,B 0,C 180,E1 -24758.713,E2 -24758.713} C_VEL
LIN {X 0,Y 139.786,Z 523.341,A -85,B 0,C 180,E1 -24761.594,E2 -24761.594} C_VEL
LIN {X 0,Y 141.466,Z 520.551,A -85,B 0,C 180,E1 -24765.85,E2 -24765.85} C_VEL
LIN {X 0,Y 144.063,Z 516.689,A -85,B 0,C 180,E1 -24769.96,E2 -24769.96} C_VEL
LIN {X 0,Y 147.314,Z 511.664,A -85,B 0,C 180,E1 -24773.916,E2 -24773.916} C_VEL
LIN {X 0,Y 150.843,Z 505.371,A -85,B 0,C 180,E1 -24777.761,E2 -24777.761} C_VEL
LIN {X 0,Y 154.784,Z 497.549,A -85,B 0,C 180,E1 -24781.469,E2 -24781.469} C_VEL
LIN {X 0,Y 158.522,Z 489.507,A -85,B 0,C 180,E1 -24784.412,E2 -24784.412} C_VEL
LIN {X 0,Y 162.066,Z 480.704,A -85,B 0,C 180,E1 -24786.983,E2 -24786.983} C_VEL
LIN {X 0,Y 165.806,Z 469.745,A -85,B 0,C 180,E1 -24789.471,E2 -24789.471} C_VEL
LIN {X 0,Y 168.558,Z 460.818,A -85,B 0,C 180,E1 -24791.002,E2 -24791.002} C_VEL
LIN {X 0,Y 168.544,Z 457.413,A -85,B 0,C 180,E1 -24791.84,E2 -24791.84} C_VEL
LIN {X 0,Y 166.762,Z 445.924,A -85,B 0,C 180,E1 -24794.84,E2 -24794.84} C_VEL
LIN {X 0,Y 164.251,Z 436.455,A -85,B 0,C 180,E1 -24797.317,E2 -24797.317} C_VEL
LIN {X 0,Y 160.01,Z 427.927,A -85,B 0,C 180,E1 -24800.133,E2 -24800.133} C_VEL
LIN {X 0,Y 155.417,Z 420.217,A -85,B 0,C 180,E1 -24802.986,E2 -24802.986} C_VEL
LIN {X 0,Y 155.203,Z 416.203,A -85,B 0,C 180,E1 -24807.084,E2 -24807.084} C_VEL
LIN {X 0,Y 154.981,Z 412.77,A -85,B 0,C 180,E1 -24811.005,E2 -24811.005} C_VEL
LIN {X 0,Y 154.832,Z 411.038,A -85,B 0,C 180,E1 -24813.004,E2 -24813.004} C_VEL
LIN {X 0,Y 154.328,Z 407.199,A -85,B 0,C 180,E1 -24818.633,E2 -24818.633} C_VEL
LIN {X 0,Y 154.125,Z 404.215,A -85,B 0,C 180,E1 -24824.121,E2 -24824.121} C_VEL
LIN {X 0,Y 154.35,Z 402.051,A -85,B 0,C 180,E1 -24829.505,E2 -24829.505} C_VEL
LIN {X 0,Y 154.408,Z 401.127,A -85,B 0,C 180,E1 -24832.151,E2 -24832.151} C_VEL
LIN {X 0,Y 155.232,Z 399.755,A -85,B 0,C 180,E1 -24839.999,E2 -24839.999} C_VEL
LIN {X 0,Y 155.51,Z 399.978,A -85,B 0,C 180,E1 -24842.589,E2 -24842.589} C_VEL
LIN {X 0,Y 155.306,Z 401.186,A -85,B 0,C 180,E1 -24845.484,E2 -24845.484} C_VEL
LIN {X 0,Y 155.051,Z 404.316,A -85,B 0,C 180,E1 -24850.445,E2 -24850.445} C_VEL
LIN {X 0,Y 155.416,Z 408.473,A -85,B 0,C 180,E1 -24855.742,E2 -24855.742} C_VEL
LIN {X 0,Y 155.964,Z 412.43,A -85,B 0,C 180,E1 -24859.615,E2 -24859.615} C_VEL
LIN {X 0,Y 156.869,Z 417.413,A -85,B 0,C 180,E1 -24863.778,E2 -24863.778} C_VEL
LIN {X 0,Y 157.987,Z 423.298,A -85,B 0,C 180,E1 -24867.843,E2 -24867.843} C_VEL
LIN {X 0,Y 160.368,Z 433.582,A -85,B 0,C 180,E1 -24873.894,E2 -24873.894} C_VEL
LIN {X 0,Y 160.741,Z 436.304,A -85,B 0,C 180,E1 -24875.206,E2 -24875.206} C_VEL
LIN {X 0,Y 161.321,Z 444.636,A -85,B 0,C 180,E1 -24878.724,E2 -24878.724} C_VEL
LIN {X 0,Y 160.824,Z 447.474,A -85,B 0,C 180,E1 -24879.621,E2 -24879.621} C_VEL
LIN {X 0,Y 161.879,Z 460.576,A -85,B 0,C 180,E1 -24880.993,E2 -24880.993} C_VEL
LIN {X 0,Y 162.624,Z 473.161,A -85,B 0,C 180,E1 -24882.695,E2 -24882.695} C_VEL
LIN {X 0,Y 162.723,Z 480.872,A -85,B 0,C 180,E1 -24883.901,E2 -24883.901} C_VEL
LIN {X 0,Y 160.379,Z 491.875,A -85,B 0,C 180,E1 -24885.22,E2 -24885.22} C_VEL
LIN {X 0,Y 157.377,Z 503.445,A -85,B 0,C 180,E1 -24887.086,E2 -24887.086} C_VEL
LIN {X 0,Y 154.211,Z 513.213,A -85,B 0,C 180,E1 -24889.08,E2 -24889.08} C_VEL
LIN {X 0,Y 150.634,Z 523.528,A -85,B 0,C 180,E1 -24891.825,E2 -24891.825} C_VEL
LIN {X 0,Y 147.043,Z 532.863,A -85,B 0,C 180,E1 -24895.011,E2 -24895.011} C_VEL
LIN {X 0,Y 143.289,Z 542.003,A -85,B 0,C 180,E1 -24899.011,E2 -24899.011} C_VEL
LIN {X 0,Y 140.324,Z 549.404,A -85,B 0,C 180,E1 -24903.216,E2 -24903.216} C_VEL
LIN {X 0,Y 138.178,Z 555.368,A -85,B 0,C 180,E1 -24907.584,E2 -24907.584} C_VEL
LIN {X 0,Y 136.729,Z 560.099,A -85,B 0,C 180,E1 -24912.045,E2 -24912.045} C_VEL
LIN {X 0,Y 135.97,Z 563.721,A -85,B 0,C 180,E1 -24916.558,E2 -24916.558} C_VEL
LIN {X 0,Y 135.896,Z 566.325,A -85,B 0,C 180,E1 -24921.082,E2 -24921.082} C_VEL
LIN {X 0,Y 136.081,Z 567.489,A -85,B 0,C 180,E1 -24924.079,E2 -24924.079} C_VEL
LIN {X 0,Y 136.345,Z 568.221,A -85,B 0,C 180,E1 -24927.053,E2 -24927.053} C_VEL
LIN {X 0,Y 136.863,Z 568.54,A -85,B 0,C 180,E1 -24930.007,E2 -24930.007} C_VEL
LIN {X 0,Y 136.457,Z 568.223,A -85,B 0,C 180,E1 -24932.959,E2 -24932.959} C_VEL
LIN {X 0,Y 136.169,Z 567.479,A -85,B 0,C 180,E1 -24935.932,E2 -24935.932} C_VEL
LIN {X 0,Y 136.027,Z 565.231,A -85,B 0,C 180,E1 -24940.996,E2 -24940.996} C_VEL
LIN {X 0,Y 136.163,Z 563.922,A -85,B 0,C 180,E1 -24943.438,E2 -24943.438} C_VEL
LIN {X 0,Y 137.316,Z 563.296,A -85,B 0,C 180,E1 -24951.001,E2 -24951.001} C_VEL
LIN {X 0,Y 141.709,Z 561.119,A -85,B 0,C 180,E1 -24959.739,E2 -24959.739} C_VEL
LIN {X 0,Y 149.423,Z 557.629,A -85,B 0,C 180,E1 -24967.701,E2 -24967.701} C_VEL
LIN {X 0,Y 158.665,Z 553.665,A -85,B 0,C 180,E1 -24973.801,E2 -24973.801} C_VEL
LIN {X 0,Y 160.251,Z 552.749,A -85,B 0,C 180,E1 -24975.074,E2 -24975.074} C_VEL
LIN {X 0,Y 162.978,Z 549.601,A -85,B 0,C 180,E1 -24979.626,E2 -24979.626} C_VEL
LIN {X 0,Y 164.966,Z 548.611,A -85,B 0,C 180,E1 -24980.778,E2 -24980.778} C_VEL
LIN {X 0,Y 170.173,Z 546.637,A -85,B 0,C 180,E1 -24982.695,E2 -24982.695} C_VEL
LIN {X 0,Y 171.057,Z 546.065,A -85,B 0,C 180,E1 -24983.388,E2 -24983.388} C_VEL
LIN {X 0,Y 159.581,Z 545.118,A -85,B 0,C 180,E1 -24988.098,E2 -24988.098} C_VEL
LIN {X 0,Y 151.559,Z 543.301,A -85,B 0,C 180,E1 -24992.374,E2 -24992.374} C_VEL
LIN {X 0,Y 144.697,Z 540.477,A -85,B 0,C 180,E1 -24997.136,E2 -24997.136} C_VEL
LIN {X 0,Y 139.154,Z 536.557,A -85,B 0,C 180,E1 -25002.361,E2 -25002.361} C_VEL
LIN {X 0,Y 134.849,Z 531.461,A -85,B 0,C 180,E1 -25007.968,E2 -25007.968} C_VEL
LIN {X 0,Y 131.807,Z 525.068,A -85,B 0,C 180,E1 -25013.88,E2 -25013.88} C_VEL
LIN {X 0,Y 130.175,Z 517.206,A -85,B 0,C 180,E1 -25020.001,E2 -25020.001} C_VEL
LIN {X 0,Y 129.847,Z 508.957,A -85,B 0,C 180,E1 -25025.436,E2 -25025.436} C_VEL
LIN {X 0,Y 130.281,Z 499.239,A -85,B 0,C 180,E1 -25030.884,E2 -25030.884} C_VEL
LIN {X 0,Y 131.351,Z 491.233,A -85,B 0,C 180,E1 -25034.724,E2 -25034.724} C_VEL
LIN {X 0,Y 133.447,Z 478.221,A -85,B 0,C 180,E1 -25040.02,E2 -25040.02} C_VEL
LIN {X 0,Y 135.903,Z 465.053,A -85,B 0,C 180,E1 -25044.439,E2 -25044.439} C_VEL
LIN {X 0,Y 138.795,Z 450.79,A -85,B 0,C 180,E1 -25048.342,E2 -25048.342} C_VEL
LIN {X 0,Y 141.064,Z 439.741,A -85,B 0,C 180,E1 -25050.969,E2 -25050.969} C_VEL
LIN {X 0,Y 141.484,Z 440.163,A -85,B 0,C 180,E1 -25051.362,E2 -25051.362} C_VEL
LIN {X 0,Y 142.944,Z 439.541,A -85,B 0,C 180,E1 -25052.266,E2 -25052.266} C_VEL
LIN {X 0,Y 145.476,Z 436.743,A -85,B 0,C 180,E1 -25053.471,E2 -25053.471} C_VEL
LIN {X 0,Y 148.997,Z 431.672,A -85,B 0,C 180,E1 -25054.886,E2 -25054.886} C_VEL
LIN {X 0,Y 151.629,Z 430.445,A -85,B 0,C 180,E1 -25056.227,E2 -25056.227} C_VEL
LIN {X 0,Y 154.421,Z 430.624,A -85,B 0,C 180,E1 -25057.704,E2 -25057.704} C_VEL
LIN {X 0,Y 155.409,Z 431.807,A -85,B 0,C 180,E1 -25058.347,E2 -25058.347} C_VEL
LIN {X 0,Y 158.517,Z 437.836,A -85,B 0,C 180,E1 -25060.632,E2 -25060.632} C_VEL
LIN {X 0,Y 160.132,Z 442.111,A -85,B 0,C 180,E1 -25062.025,E2 -25062.025} C_VEL
LIN {X 0,Y 162.056,Z 451.69,A -85,B 0,C 180,E1 -25064.659,E2 -25064.659} C_VEL
LIN {X 0,Y 163.091,Z 460.363,A -85,B 0,C 180,E1 -25067.104,E2 -25067.104} C_VEL
LIN {X 0,Y 163.096,Z 462.078,A -85,B 0,C 180,E1 -25067.556,E2 -25067.556} C_VEL
LIN {X 0,Y 159.72,Z 472.821,A -85,B 0,C 180,E1 -25069.525,E2 -25069.525} C_VEL
LIN {X 0,Y 155.709,Z 483.312,A -85,B 0,C 180,E1 -25072.043,E2 -25072.043} C_VEL
LIN {X 0,Y 152.166,Z 491.816,A -85,B 0,C 180,E1 -25074.73,E2 -25074.73} C_VEL
LIN {X 0,Y 147.483,Z 501.096,A -85,B 0,C 180,E1 -25078.38,E2 -25078.38} C_VEL
LIN {X 0,Y 143.606,Z 508.135,A -85,B 0,C 180,E1 -25082.079,E2 -25082.079} C_VEL
LIN {X 0,Y 139.785,Z 514.299,A -85,B 0,C 180,E1 -25086.276,E2 -25086.276} C_VEL
LIN {X 0,Y 136.643,Z 518.952,A -85,B 0,C 180,E1 -25090.462,E2 -25090.462} C_VEL
LIN {X 0,Y 134.758,Z 521.477,A -85,B 0,C 180,E1 -25093.324,E2 -25093.324} C_VEL
LIN {X 0,Y 132.93,Z 524.31,A -85,B 0,C 180,E1 -25097.784,E2 -25097.784} C_VEL
LIN {X 0,Y 132.133,Z 525.663,A -85,B 0,C 180,E1 -25100.811,E2 -25100.811} C_VEL
LIN {X 0,Y 131.04,Z 527.223,A -85,B 0,C 180,E1 -25106.918,E2 -25106.918} C_VEL
LIN {X 0,Y 130.911,Z 527.446,A -85,B 0,C 180,E1 -25109.993,E2 -25109.993} C_VEL
LIN {X 0,Y 131.388,Z 526.686,A -85,B 0,C 180,E1 -25116.134,E2 -25116.134} C_VEL
LIN {X 0,Y 132.135,Z 525.729,A -85,B 0,C 180,E1 -25119.174,E2 -25119.174} C_VEL
LIN {X 0,Y 132.915,Z 524.418,A -85,B 0,C 180,E1 -25122.203,E2 -25122.203} C_VEL
LIN {X 0,Y 134.726,Z 521.626,A -85,B 0,C 180,E1 -25126.665,E2 -25126.665} C_VEL
LIN {X 0,Y 137.488,Z 517.763,A -85,B 0,C 180,E1 -25130.958,E2 -25130.958} C_VEL
LIN {X 0,Y 140.929,Z 512.737,A -85,B 0,C 180,E1 -25135.072,E2 -25135.072} C_VEL
LIN {X 0,Y 144.684,Z 506.44,A -85,B 0,C 180,E1 -25139.053,E2 -25139.053} C_VEL
LIN {X 0,Y 148.853,Z 498.617,A -85,B 0,C 180,E1 -25142.877,E2 -25142.877} C_VEL
LIN {X 0,Y 152.786,Z 490.573,A -85,B 0,C 180,E1 -25145.899,E2 -25145.899} C_VEL
LIN {X 0,Y 156.515,Z 481.766,A -85,B 0,C 180,E1 -25148.529,E2 -25148.529} C_VEL
LIN {X 0,Y 160.449,Z 470.802,A -85,B 0,C 180,E1 -25151.064,E2 -25151.064} C_VEL
LIN {X 0,Y 163.115,Z 462.658,A -85,B 0,C 180,E1 -25152.491,E2 -25152.491} C_VEL
LIN {X 0,Y 163.022,Z 458.533,A -85,B 0,C 180,E1 -25153.603,E2 -25153.603} C_VEL
LIN {X 0,Y 161.645,Z 448.46,A -85,B 0,C 180,E1 -25156.395,E2 -25156.395} C_VEL
LIN {X 0,Y 159.772,Z 440.625,A -85,B 0,C 180,E1 -25158.609,E2 -25158.609} C_VEL
LIN {X 0,Y 155.978,Z 432.585,A -85,B 0,C 180,E1 -25161.51,E2 -25161.51} C_VEL
LIN {X 0,Y 151.846,Z 425.321,A -85,B 0,C 180,E1 -25164.426,E2 -25164.426} C_VEL
LIN {X 0,Y 149.569,Z 421.6,A -85,B 0,C 180,E1 -25166.072,E2 -25166.072} C_VEL
LIN {X 0,Y 149.423,Z 417.823,A -85,B 0,C 180,E1 -25170.404,E2 -25170.404} C_VEL
LIN {X 0,Y 149.393,Z 415.505,A -85,B 0,C 180,E1 -25173.341,E2 -25173.341} C_VEL
LIN {X 0,Y 148.993,Z 412.5,A -85,B 0,C 180,E1 -25177.829,E2 -25177.829} C_VEL
LIN {X 0,Y 148.961,Z 409.422,A -85,B 0,C 180,E1 -25183.555,E2 -25183.555} C_VEL
LIN {X 0,Y 149.136,Z 407.097,A -85,B 0,C 180,E1 -25189.134,E2 -25189.134} C_VEL
LIN {X 0,Y 149.419,Z 406.351,A -85,B 0,C 180,E1 -25191.887,E2 -25191.887} C_VEL
LIN {X 0,Y 149.865,Z 405.337,A -85,B 0,C 180,E1 -25197.311,E2 -25197.311} C_VEL
LIN {X 0,Y 150.422,Z 405.028,A -85,B 0,C 180,E1 -25199.999,E2 -25199.999} C_VEL
LIN {X 0,Y 150.767,Z 405.392,A -85,B 0,C 180,E1 -25202.671,E2 -25202.671} C_VEL
LIN {X 0,Y 150.565,Z 406.525,A -85,B 0,C 180,E1 -25205.356,E2 -25205.356} C_VEL
LIN {X 0,Y 150.288,Z 410.116,A -85,B 0,C 180,E1 -25210.918,E2 -25210.918} C_VEL
LIN {X 0,Y 150.724,Z 414.473,A -85,B 0,C 180,E1 -25216.245,E2 -25216.245} C_VEL
LIN {X 0,Y 151.682,Z 420.877,A -85,B 0,C 180,E1 -25222.098,E2 -25222.098} C_VEL
LIN {X 0,Y 152.692,Z 427.013,A -85,B 0,C 180,E1 -25226.663,E2 -25226.663} C_VEL
LIN {X 0,Y 155.111,Z 438.836,A -85,B 0,C 180,E1 -25233.813,E2 -25233.813} C_VEL
LIN {X 0,Y 155.473,Z 446.665,A -85,B 0,C 180,E1 -25237.199,E2 -25237.199} C_VEL
LIN {X 0,Y 156.29,Z 449.759,A -85,B 0,C 180,E1 -25237.801,E2 -25237.801} C_VEL
LIN {X 0,Y 157.072,Z 462.399,A -85,B 0,C 180,E1 -25239.238,E2 -25239.238} C_VEL
LIN {X 0,Y 157.488,Z 474.629,A -85,B 0,C 180,E1 -25241.034,E2 -25241.034} C_VEL
LIN {X 0,Y 157.463,Z 481.311,A -85,B 0,C 180,E1 -25242.155,E2 -25242.155} C_VEL
LIN {X 0,Y 155.028,Z 492.02,A -85,B 0,C 180,E1 -25243.513,E2 -25243.513} C_VEL
LIN {X 0,Y 151.688,Z 503.902,A -85,B 0,C 180,E1 -25245.522,E2 -25245.522} C_VEL
LIN {X 0,Y 148.374,Z 513.388,A -85,B 0,C 180,E1 -25247.558,E2 -25247.558} C_VEL
LIN {X 0,Y 144.184,Z 524.42,A -85,B 0,C 180,E1 -25250.689,E2 -25250.689} C_VEL
LIN {X 0,Y 140.431,Z 533.43,A -85,B 0,C 180,E1 -25253.992,E2 -25253.992} C_VEL
LIN {X 0,Y 136.502,Z 542.231,A -85,B 0,C 180,E1 -25258.157,E2 -25258.157} C_VEL
LIN {X 0,Y 133.36,Z 549.461,A -85,B 0,C 180,E1 -25262.635,E2 -25262.635} C_VEL
LIN {X 0,Y 130.86,Z 555.98,A -85,B 0,C 180,E1 -25267.926,E2 -25267.926} C_VEL
LIN {X 0,Y 129.488,Z 560.336,A -85,B 0,C 180,E1 -25272.64,E2 -25272.64} C_VEL
LIN {X 0,Y 128.859,Z 563.613,A -85,B 0,C 180,E1 -25277.407,E2 -25277.407} C_VEL
LIN {X 0,Y 128.825,Z 565.227,A -85,B 0,C 180,E1 -25280.588,E2 -25280.588} C_VEL
LIN {X 0,Y 129.02,Z 566.4,A -85,B 0,C 180,E1 -25283.753,E2 -25283.753} C_VEL
LIN {X 0,Y 129.28,Z 567.135,A -85,B 0,C 180,E1 -25286.891,E2 -25286.891} C_VEL
LIN {X 0,Y 129.828,Z 567.46,A -85,B 0,C 180,E1 -25290.008,E2 -25290.008} C_VEL
LIN {X 0,Y 129.388,Z 567.137,A -85,B 0,C 180,E1 -25293.121,E2 -25293.121} C_VEL
LIN {X 0,Y 129.105,Z 566.389,A -85,B 0,C 180,E1 -25296.258,E2 -25296.258} C_VEL
LIN {X 0,Y 128.964,Z 564.33,A -85,B 0,C 180,E1 -25301.215,E2 -25301.215} C_VEL
LIN {X 0,Y 129.412,Z 561.947,A -85,B 0,C 180,E1 -25305.359,E2 -25305.359} C_VEL
LIN {X 0,Y 131.812,Z 561.068,A -85,B 0,C 180,E1 -25314.989,E2 -25314.989} C_VEL
LIN {X 0,Y 137.893,Z 558.687,A -85,B 0,C 180,E1 -25324.107,E2 -25324.107} C_VEL
LIN {X 0,Y 147.276,Z 555.177,A -85,B 0,C 180,E1 -25331.927,E2 -25331.927} C_VEL
LIN {X 0,Y 160.265,Z 550.376,A -85,B 0,C 180,E1 -25338.87,E2 -25338.87} C_VEL
LIN {X 0,Y 164.966,Z 548.611,A -85,B 0,C 180,E1 -25340.778,E2 -25340.778} C_VEL
LIN {X 0,Y 165.602,Z 548.106,A -85,B 0,C 180,E1 -25341.48,E2 -25341.48} C_VEL
LIN {X 0,Y 164.874,Z 547.638,A -85,B 0,C 180,E1 -25342.462,E2 -25342.462} C_VEL
LIN {X 0,Y 163.155,Z 547.334,A -85,B 0,C 180,E1 -25343.412,E2 -25343.412} C_VEL
LIN {X 0,Y 152.946,Z 546.263,A -85,B 0,C 180,E1 -25347.066,E2 -25347.066} C_VEL
LIN {X 0,Y 145.381,Z 544.289,A -85,B 0,C 180,E1 -25351.092,E2 -25351.092} C_VEL
LIN {X 0,Y 138.207,Z 541.111,A -85,B 0,C 180,E1 -25355.997,E2 -25355.997} C_VEL
LIN {X 0,Y 132.408,Z 536.85,A -85,B 0,C 180,E1 -25361.431,E2 -25361.431} C_VEL
LIN {X 0,Y 127.927,Z 531.441,A -85,B 0,C 180,E1 -25367.307,E2 -25367.307} C_VEL
LIN {X 0,Y 124.743,Z 524.729,A -85,B 0,C 180,E1 -25373.531,E2 -25373.531} C_VEL
LIN {X 0,Y 123.066,Z 516.551,A -85,B 0,C 180,E1 -25380.001,E2 -25380.001} C_VEL
LIN {X 0,Y 122.766,Z 508.045,A -85,B 0,C 180,E1 -25385.751,E2 -25385.751} C_VEL
LIN {X 0,Y 123.335,Z 497.967,A -85,B 0,C 180,E1 -25391.506,E2 -25391.506} C_VEL
LIN {X 0,Y 124.453,Z 489.729,A -85,B 0,C 180,E1 -25395.561,E2 -25395.561} C_VEL
LIN {X 0,Y 126.757,Z 476.271,A -85,B 0,C 180,E1 -25401.126,E2 -25401.126} C_VEL
LIN {X 0,Y 129.632,Z 461.399,A -85,B 0,C 180,E1 -25406.137,E2 -25406.137} C_VEL
LIN {X 0,Y 130.32,Z 458.208,A -85,B 0,C 180,E1 -25407.176,E2 -25407.176} C_VEL
LIN {X 0,Y 131.988,Z 457.872,A -85,B 0,C 180,E1 -25408.636,E2 -25408.636} C_VEL
LIN {X 0,Y 135.331,Z 454.749,A -85,B 0,C 180,E1 -25410.421,E2 -25410.421} C_VEL
LIN {X 0,Y 139.491,Z 449.44,A -85,B 0,C 180,E1 -25412.047,E2 -25412.047} C_VEL
LIN {X 0,Y 141.12,Z 446.892,A -85,B 0,C 180,E1 -25412.582,E2 -25412.582} C_VEL
LIN {X 0,Y 143.858,Z 445.123,A -85,B 0,C 180,E1 -25414.015,E2 -25414.015} C_VEL
LIN {X 0,Y 147.192,Z 441.615,A -85,B 0,C 180,E1 -25415.377,E2 -25415.377} C_VEL
LIN {X 0,Y 150.143,Z 437.944,A -85,B 0,C 180,E1 -25416.434,E2 -25416.434} C_VEL
LIN {X 0,Y 151.514,Z 437.342,A -85,B 0,C 180,E1 -25417.087,E2 -25417.087} C_VEL
LIN {X 0,Y 152.086,Z 437.647,A -85,B 0,C 180,E1 -25417.444,E2 -25417.444} C_VEL
LIN {X 0,Y 155.095,Z 444.344,A -85,B 0,C 180,E1 -25420.115,E2 -25420.115} C_VEL
LIN {X 0,Y 156.712,Z 452.367,A -85,B 0,C 180,E1 -25422.532,E2 -25422.532} C_VEL
LIN {X 0,Y 157.737,Z 462.909,A -85,B 0,C 180,E1 -25425.67,E2 -25425.67} C_VEL
LIN {X 0,Y 157.657,Z 464.283,A -85,B 0,C 180,E1 -25426.021,E2 -25426.021} C_VEL
LIN {X 0,Y 153.979,Z 475.155,A -85,B 0,C 180,E1 -25428.117,E2 -25428.117} C_VEL
LIN {X 0,Y 149.345,Z 486.44,A -85,B 0,C 180,E1 -25430.986,E2 -25430.986} C_VEL
LIN {X 0,Y 145.577,Z 494.621,A -85,B 0,C 180,E1 -25433.737,E2 -25433.737} C_VEL
LIN {X 0,Y 141.552,Z 502.172,A -85,B 0,C 180,E1 -25436.89,E2 -25436.89} C_VEL
LIN {X 0,Y 137.464,Z 509.208,A -85,B 0,C 180,E1 -25440.714,E2 -25440.714} C_VEL
LIN {X 0,Y 133.391,Z 515.375,A -85,B 0,C 180,E1 -25445.063,E2 -25445.063} C_VEL
LIN {X 0,Y 130.054,Z 520.028,A -85,B 0,C 180,E1 -25449.428,E2 -25449.428} C_VEL
LIN {X 0,Y 128.05,Z 522.554,A -85,B 0,C 180,E1 -25452.423,E2 -25452.423} C_VEL
LIN {X 0,Y 126.078,Z 525.388,A -85,B 0,C 180,E1 -25457.109,E2 -25457.109} C_VEL
LIN {X 0,Y 125.213,Z 526.74,A -85,B 0,C 180,E1 -25460.298,E2 -25460.298} C_VEL
LIN {X 0,Y 124.048,Z 528.298,A -85,B 0,C 180,E1 -25466.744,E2 -25466.744} C_VEL
LIN {X 0,Y 123.905,Z 528.521,A -85,B 0,C 180,E1 -25469.992,E2 -25469.992} C_VEL
LIN {X 0,Y 124.432,Z 527.76,A -85,B 0,C 180,E1 -25476.478,E2 -25476.478} C_VEL
LIN {X 0,Y 125.213,Z 526.806,A -85,B 0,C 180,E1 -25479.686,E2 -25479.686} C_VEL
LIN {X 0,Y 126.062,Z 525.494,A -85,B 0,C 180,E1 -25482.877,E2 -25482.877} C_VEL
LIN {X 0,Y 128.017,Z 522.702,A -85,B 0,C 180,E1 -25487.566,E2 -25487.566} C_VEL
LIN {X 0,Y 130.959,Z 518.837,A -85,B 0,C 180,E1 -25492.056,E2 -25492.056} C_VEL
LIN {X 0,Y 134.607,Z 513.809,A -85,B 0,C 180,E1 -25496.338,E2 -25496.338} C_VEL
LIN {X 0,Y 138.607,Z 507.509,A -85,B 0,C 180,E1 -25500.458,E2 -25500.458} C_VEL
LIN {X 0,Y 143.014,Z 499.685,A -85,B 0,C 180,E1 -25504.402,E2 -25504.402} C_VEL
LIN {X 0,Y 147.158,Z 491.64,A -85,B 0,C 180,E1 -25507.502,E2 -25507.502} C_VEL
LIN {X 0,Y 151.095,Z 482.827,A -85,B 0,C 180,E1 -25510.184,E2 -25510.184} C_VEL
LIN {X 0,Y 155.225,Z 471.86,A -85,B 0,C 180,E1 -25512.767,E2 -25512.767} C_VEL
LIN {X 0,Y 157.88,Z 463.752,A -85,B 0,C 180,E1 -25514.252,E2 -25514.252} C_VEL
LIN {X 0,Y 157.062,Z 453.851,A -85,B 0,C 180,E1 -25517.194,E2 -25517.194} C_VEL
LIN {X 0,Y 155.368,Z 445.022,A -85,B 0,C 180,E1 -25519.864,E2 -25519.864} C_VEL
LIN {X 0,Y 152.159,Z 437.522,A -85,B 0,C 180,E1 -25522.785,E2 -25522.785} C_VEL
LIN {X 0,Y 148.501,Z 430.54,A -85,B 0,C 180,E1 -25525.794,E2 -25525.794} C_VEL
LIN {X 0,Y 146.046,Z 426.604,A -85,B 0,C 180,E1 -25527.753,E2 -25527.753} C_VEL
LIN {X 0,Y 143.87,Z 423.051,A -85,B 0,C 180,E1 -25529.648,E2 -25529.648} C_VEL
LIN {X 0,Y 143.876,Z 419.762,A -85,B 0,C 180,E1 -25533.919,E2 -25533.919} C_VEL
LIN {X 0,Y 143.629,Z 416.145,A -85,B 0,C 180,E1 -25539.968,E2 -25539.968} C_VEL
LIN {X 0,Y 143.746,Z 414.681,A -85,B 0,C 180,E1 -25542.94,E2 -25542.94} C_VEL
LIN {X 0,Y 144.096,Z 412.333,A -85,B 0,C 180,E1 -25548.749,E2 -25548.749} C_VEL
LIN {X 0,Y 144.342,Z 411.476,A -85,B 0,C 180,E1 -25551.6,E2 -25551.6} C_VEL
LIN {X 0,Y 144.952,Z 410.504,A -85,B 0,C 180,E1 -25557.22,E2 -25557.22} C_VEL
LIN {X 0,Y 145.568,Z 410.235,A -85,B 0,C 180,E1 -25559.999,E2 -25559.999} C_VEL
LIN {X 0,Y 145.854,Z 410.677,A -85,B 0,C 180,E1 -25562.761,E2 -25562.761} C_VEL
LIN {X 0,Y 145.673,Z 411.986,A -85,B 0,C 180,E1 -25565.536,E2 -25565.536} C_VEL
LIN {X 0,Y 145.517,Z 415.738,A -85,B 0,C 180,E1 -25571.138,E2 -25571.138} C_VEL
LIN {X 0,Y 145.853,Z 419.282,A -85,B 0,C 180,E1 -25575.513,E2 -25575.513} C_VEL
LIN {X 0,Y 146.588,Z 425.115,A -85,B 0,C 180,E1 -25581.073,E2 -25581.073} C_VEL
LIN {X 0,Y 147.548,Z 431.785,A -85,B 0,C 180,E1 -25586.141,E2 -25586.141} C_VEL
LIN {X 0,Y 149.446,Z 442.19,A -85,B 0,C 180,E1 -25592.736,E2 -25592.736} C_VEL
LIN {X 0,Y 149.593,Z 445.222,A -85,B 0,C 180,E1 -25594.112,E2 -25594.112} C_VEL
LIN {X 0,Y 151.916,Z 452.008,A -85,B 0,C 180,E1 -25595.873,E2 -25595.873} C_VEL
LIN {X 0,Y 152.408,Z 464.738,A -85,B 0,C 180,E1 -25597.451,E2 -25597.451} C_VEL
LIN {X 0,Y 152.429,Z 476.64,A -85,B 0,C 180,E1 -25599.341,E2 -25599.341} C_VEL
LIN {X 0,Y 152.219,Z 482.786,A -85,B 0,C 180,E1 -25600.457,E2 -25600.457} C_VEL
LIN {X 0,Y 149.116,Z 494.629,A -85,B 0,C 180,E1 -25602.082,E2 -25602.082} C_VEL
LIN {X 0,Y 145.63,Z 505.689,A -85,B 0,C 180,E1 -25604.133,E2 -25604.133} C_VEL
LIN {X 0,Y 142.195,Z 514.678,A -85,B 0,C 180,E1 -25606.226,E2 -25606.226} C_VEL
LIN {X 0,Y 137.924,Z 525.006,A -85,B 0,C 180,E1 -25609.348,E2 -25609.348} C_VEL
LIN {X 0,Y 133.864,Z 533.926,A -85,B 0,C 180,E1 -25612.87,E2 -25612.87} C_VEL
LIN {X 0,Y 129.749,Z 542.403,A -85,B 0,C 180,E1 -25617.213,E2 -25617.213} C_VEL
LIN {X 0,Y 126.515,Z 549.308,A -85,B 0,C 180,E1 -25621.834,E2 -25621.834} C_VEL
LIN {X 0,Y 124.151,Z 554.867,A -85,B 0,C 180,E1 -25626.665,E2 -25626.665} C_VEL
LIN {X 0,Y 122.597,Z 559.227,A -85,B 0,C 180,E1 -25631.63,E2 -25631.63} C_VEL
LIN {X 0,Y 121.829,Z 562.507,A -85,B 0,C 180,E1 -25636.667,E2 -25636.667} C_VEL
LIN {X 0,Y 121.768,Z 564.129,A -85,B 0,C 180,E1 -25640.037,E2 -25640.037} C_VEL
LIN {X 0,Y 121.938,Z 565.307,A -85,B 0,C 180,E1 -25643.389,E2 -25643.389} C_VEL
LIN {X 0,Y 122.212,Z 566.049,A -85,B 0,C 180,E1 -25646.711,E2 -25646.711} C_VEL
LIN {X 0,Y 122.791,Z 566.38,A -85,B 0,C 180,E1 -25650.008,E2 -25650.008} C_VEL
LIN {X 0,Y 122.317,Z 566.05,A -85,B 0,C 180,E1 -25653.302,E2 -25653.302} C_VEL
LIN {X 0,Y 122.042,Z 565.298,A -85,B 0,C 180,E1 -25656.622,E2 -25656.622} C_VEL
LIN {X 0,Y 121.93,Z 563.4,A -85,B 0,C 180,E1 -25661.521,E2 -25661.521} C_VEL
LIN {X 0,Y 122.786,Z 559.89,A -85,B 0,C 180,E1 -25667.495,E2 -25667.495} C_VEL
LIN {X 0,Y 125.538,Z 559.176,A -85,B 0,C 180,E1 -25676.615,E2 -25676.615} C_VEL
LIN {X 0,Y 132.026,Z 557.155,A -85,B 0,C 180,E1 -25685.85,E2 -25685.85} C_VEL
LIN {X 0,Y 142.017,Z 554.025,A -85,B 0,C 180,E1 -25693.862,E2 -25693.862} C_VEL
LIN {X 0,Y 155.059,Z 549.809,A -85,B 0,C 180,E1 -25700.615,E2 -25700.615} C_VEL
LIN {X 0,Y 160.682,Z 547.997,A -85,B 0,C 180,E1 -25702.823,E2 -25702.823} C_VEL
LIN {X 0,Y 161.204,Z 547.5,A -85,B 0,C 180,E1 -25703.573,E2 -25703.573} C_VEL
LIN {X 0,Y 152.946,Z 546.263,A -85,B 0,C 180,E1 -25707.066,E2 -25707.066} C_VEL
LIN {X 0,Y 148.879,Z 545.597,A -85,B 0,C 180,E1 -25708.67,E2 -25708.67} C_VEL
LIN {X 0,Y 141.137,Z 544.29,A -85,B 0,C 180,E1 -25711.066,E2 -25711.066} C_VEL
LIN {X 0,Y 133.838,Z 542.417,A -85,B 0,C 180,E1 -25713.731,E2 -25713.731} C_VEL
LIN {X 0,Y 130.566,Z 540.832,A -85,B 0,C 180,E1 -25715.747,E2 -25715.747} C_VEL
LIN {X 0,Y 124.409,Z 535.706,A -85,B 0,C 180,E1 -25721.9,E2 -25721.9} C_VEL
LIN {X 0,Y 120.098,Z 529.676,A -85,B 0,C 180,E1 -25728.183,E2 -25728.183} C_VEL
LIN {X 0,Y 116.912,Z 521.29,A -85,B 0,C 180,E1 -25735.692,E2 -25735.692} C_VEL
LIN {X 0,Y 115.736,Z 512.164,A -85,B 0,C 180,E1 -25742.612,E2 -25742.612} C_VEL
LIN {X 0,Y 115.825,Z 502.719,A -85,B 0,C 180,E1 -25748.727,E2 -25748.727} C_VEL
LIN {X 0,Y 117.318,Z 490.147,A -85,B 0,C 180,E1 -25755.457,E2 -25755.457} C_VEL
LIN {X 0,Y 119.516,Z 477.381,A -85,B 0,C 180,E1 -25761.112,E2 -25761.112} C_VEL
LIN {X 0,Y 120.581,Z 471.715,A -85,B 0,C 180,E1 -25763.282,E2 -25763.282} C_VEL
LIN {X 0,Y 121.021,Z 471.859,A -85,B 0,C 180,E1 -25763.987,E2 -25763.987} C_VEL
LIN {X 0,Y 122.564,Z 471.169,A -85,B 0,C 180,E1 -25765.473,E2 -25765.473} C_VEL
LIN {X 0,Y 124.643,Z 469.475,A -85,B 0,C 180,E1 -25766.814,E2 -25766.814} C_VEL
LIN {X 0,Y 129.58,Z 464.453,A -85,B 0,C 180,E1 -25769.219,E2 -25769.219} C_VEL
LIN {X 0,Y 131.501,Z 463.489,A -85,B 0,C 180,E1 -25770.514,E2 -25770.514} C_VEL
LIN {X 0,Y 135.081,Z 460.487,A -85,B 0,C 180,E1 -25772.229,E2 -25772.229} C_VEL
LIN {X 0,Y 139.202,Z 455.971,A -85,B 0,C 180,E1 -25773.737,E2 -25773.737} C_VEL
LIN {X 0,Y 141.305,Z 453.261,A -85,B 0,C 180,E1 -25774.372,E2 -25774.372} C_VEL
LIN {X 0,Y 147.039,Z 448.403,A -85,B 0,C 180,E1 -25776.689,E2 -25776.689} C_VEL
LIN {X 0,Y 149.457,Z 445.658,A -85,B 0,C 180,E1 -25777.473,E2 -25777.473} C_VEL
LIN {X 0,Y 150.939,Z 449.489,A -85,B 0,C 180,E1 -25779.094,E2 -25779.094} C_VEL
LIN {X 0,Y 152.151,Z 458.88,A -85,B 0,C 180,E1 -25782.052,E2 -25782.052} C_VEL
LIN {X 0,Y 152.503,Z 465.698,A -85,B 0,C 180,E1 -25784.218,E2 -25784.218} C_VEL
LIN {X 0,Y 148.827,Z 476.223,A -85,B 0,C 180,E1 -25786.312,E2 -25786.312} C_VEL
LIN {X 0,Y 143.959,Z 487.512,A -85,B 0,C 180,E1 -25789.227,E2 -25789.227} C_VEL
LIN {X 0,Y 139.99,Z 495.692,A -85,B 0,C 180,E1 -25792.041,E2 -25792.041} C_VEL
LIN {X 0,Y 135.726,Z 503.247,A -85,B 0,C 180,E1 -25795.27,E2 -25795.27} C_VEL
LIN {X 0,Y 130.646,Z 511.406,A -85,B 0,C 180,E1 -25799.961,E2 -25799.961} C_VEL
LIN {X 0,Y 127.063,Z 516.451,A -85,B 0,C 180,E1 -25803.729,E2 -25803.729} C_VEL
LIN {X 0,Y 123.511,Z 521.105,A -85,B 0,C 180,E1 -25808.285,E2 -25808.285} C_VEL
LIN {X 0,Y 121.377,Z 523.632,A -85,B 0,C 180,E1 -25811.422,E2 -25811.422} C_VEL
LIN {X 0,Y 119.244,Z 526.466,A -85,B 0,C 180,E1 -25816.356,E2 -25816.356} C_VEL
LIN {X 0,Y 118.302,Z 527.817,A -85,B 0,C 180,E1 -25819.726,E2 -25819.726} C_VEL
LIN {X 0,Y 117.055,Z 529.373,A -85,B 0,C 180,E1 -25826.55,E2 -25826.55} C_VEL
LIN {X 0,Y 116.896,Z 529.597,A -85,B 0,C 180,E1 -25829.992,E2 -25829.992} C_VEL
LIN {X 0,Y 117.477,Z 528.834,A -85,B 0,C 180,E1 -25836.863,E2 -25836.863} C_VEL
LIN {X 0,Y 118.301,Z 527.882,A -85,B 0,C 180,E1 -25840.258,E2 -25840.258} C_VEL
LIN {X 0,Y 119.227,Z 526.57,A -85,B 0,C 180,E1 -25843.629,E2 -25843.629} C_VEL
LIN {X 0,Y 121.343,Z 523.777,A -85,B 0,C 180,E1 -25848.566,E2 -25848.566} C_VEL
LIN {X 0,Y 124.483,Z 519.911,A -85,B 0,C 180,E1 -25853.269,E2 -25853.269} C_VEL
LIN {X 0,Y 128.357,Z 514.882,A -85,B 0,C 180,E1 -25857.727,E2 -25857.727} C_VEL
LIN {X 0,Y 133.277,Z 507.517,A -85,B 0,C 180,E1 -25862.618,E2 -25862.618} C_VEL
LIN {X 0,Y 138.109,Z 499.278,A -85,B 0,C 180,E1 -25866.712,E2 -25866.712} C_VEL
LIN {X 0,Y 142.524,Z 490.873,A -85,B 0,C 180,E1 -25869.86,E2 -25869.86} C_VEL
LIN {X 0,Y 147.259,Z 480.5,A -85,B 0,C 180,E1 -25872.84,E2 -25872.84} C_VEL
LIN {X 0,Y 151.423,Z 469.514,A -85,B 0,C 180,E1 -25875.231,E2 -25875.231} C_VEL
LIN {X 0,Y 152.604,Z 465.577,A -85,B 0,C 180,E1 -25876.002,E2 -25876.002} C_VEL
LIN {X 0,Y 151.993,Z 455.778,A -85,B 0,C 180,E1 -25879.1,E2 -25879.1} C_VEL
LIN {X 0,Y 151.02,Z 449.578,A -85,B 0,C 180,E1 -25881.09,E2 -25881.09} C_VEL
LIN {X 0,Y 148.13,Z 442.011,A -85,B 0,C 180,E1 -25884.266,E2 -25884.266} C_VEL
LIN {X 0,Y 145.122,Z 435.74,A -85,B 0,C 180,E1 -25887.193,E2 -25887.193} C_VEL
LIN {X 0,Y 143.211,Z 432.375,A -85,B 0,C 180,E1 -25888.983,E2 -25888.983} C_VEL
LIN {X 0,Y 140.811,Z 428.528,A -85,B 0,C 180,E1 -25891.244,E2 -25891.244} C_VEL
LIN {X 0,Y 138.41,Z 424.607,A -85,B 0,C 180,E1 -25893.823,E2 -25893.823} C_VEL
LIN {X 0,Y 138.379,Z 421.443,A -85,B 0,C 180,E1 -25899.174,E2 -25899.174} C_VEL
LIN {X 0,Y 138.66,Z 418.609,A -85,B 0,C 180,E1 -25905.318,E2 -25905.318} C_VEL
LIN {X 0,Y 138.999,Z 417.5,A -85,B 0,C 180,E1 -25908.331,E2 -25908.331} C_VEL
LIN {X 0,Y 139.246,Z 416.613,A -85,B 0,C 180,E1 -25911.29,E2 -25911.29} C_VEL
LIN {X 0,Y 140.069,Z 415.704,A -85,B 0,C 180,E1 -25917.123,E2 -25917.123} C_VEL
LIN {X 0,Y 140.727,Z 415.466,A -85,B 0,C 180,E1 -25919.999,E2 -25919.999} C_VEL
LIN {X 0,Y 141.018,Z 416.05,A -85,B 0,C 180,E1 -25922.856,E2 -25922.856} C_VEL
LIN {X 0,Y 140.838,Z 417.5,A -85,B 0,C 180,E1 -25925.727,E2 -25925.727} C_VEL
LIN {X 0,Y 140.685,Z 421.383,A -85,B 0,C 180,E1 -25931.525,E2 -25931.525} C_VEL
LIN {X 0,Y 141.034,Z 425.206,A -85,B 0,C 180,E1 -25936.057,E2 -25936.057} C_VEL
LIN {X 0,Y 141.713,Z 431.466,A -85,B 0,C 180,E1 -25941.835,E2 -25941.835} C_VEL
LIN {X 0,Y 142.441,Z 437.554,A -85,B 0,C 180,E1 -25946.362,E2 -25946.362} C_VEL
LIN {X 0,Y 143.505,Z 443.674,A -85,B 0,C 180,E1 -25950.333,E2 -25950.333} C_VEL
LIN {X 0,Y 145.885,Z 449.185,A -85,B 0,C 180,E1 -25952.327,E2 -25952.327} C_VEL
LIN {X 0,Y 147.742,Z 455.155,A -85,B 0,C 180,E1 -25953.976,E2 -25953.976} C_VEL
LIN {X 0,Y 147.811,Z 466.638,A -85,B 0,C 180,E1 -25955.532,E2 -25955.532} C_VEL
LIN {X 0,Y 147.456,Z 478.316,A -85,B 0,C 180,E1 -25957.516,E2 -25957.516} C_VEL
LIN {X 0,Y 146.835,Z 484.928,A -85,B 0,C 180,E1 -25958.718,E2 -25958.718} C_VEL
LIN {X 0,Y 143.269,Z 496.996,A -85,B 0,C 180,E1 -25960.517,E2 -25960.517} C_VEL
LIN {X 0,Y 139.073,Z 508.635,A -85,B 0,C 180,E1 -25962.894,E2 -25962.894} C_VEL
LIN {X 0,Y 134.672,Z 519.179,A -85,B 0,C 180,E1 -25965.746,E2 -25965.746} C_VEL
LIN {X 0,Y 130.26,Z 528.541,A -85,B 0,C 180,E1 -25969.054,E2 -25969.054} C_VEL
LIN {X 0,Y 125.874,Z 537.283,A -85,B 0,C 180,E1 -25973.126,E2 -25973.126} C_VEL
LIN {X 0,Y 121.836,Z 544.928,A -85,B 0,C 180,E1 -25977.763,E2 -25977.763} C_VEL
LIN {X 0,Y 118.79,Z 550.963,A -85,B 0,C 180,E1 -25982.552,E2 -25982.552} C_VEL
LIN {X 0,Y 116.839,Z 555.313,A -85,B 0,C 180,E1 -25986.994,E2 -25986.994} C_VEL
LIN {X 0,Y 115.367,Z 559.308,A -85,B 0,C 180,E1 -25992.276,E2 -25992.276} C_VEL
LIN {X 0,Y 114.735,Z 562.678,A -85,B 0,C 180,E1 -25998.535,E2 -25998.535} C_VEL
LIN {X 0,Y 114.846,Z 564.211,A -85,B 0,C 180,E1 -26002.979,E2 -26002.979} C_VEL
LIN {X 0,Y 115.139,Z 564.962,A -85,B 0,C 180,E1 -26006.509,E2 -26006.509} C_VEL
LIN {X 0,Y 115.749,Z 565.3,A -85,B 0,C 180,E1 -26010.008,E2 -26010.008} C_VEL
LIN {X 0,Y 115.244,Z 564.962,A -85,B 0,C 180,E1 -26013.505,E2 -26013.505} C_VEL
LIN {X 0,Y 114.962,Z 564.204,A -85,B 0,C 180,E1 -26017.031,E2 -26017.031} C_VEL
LIN {X 0,Y 114.881,Z 562.49,A -85,B 0,C 180,E1 -26021.82,E2 -26021.82} C_VEL
LIN {X 0,Y 115.732,Z 559.297,A -85,B 0,C 180,E1 -26027.684,E2 -26027.684} C_VEL
LIN {X 0,Y 116.509,Z 557.714,A -85,B 0,C 180,E1 -26030.303,E2 -26030.303} C_VEL
LIN {X 0,Y 121.188,Z 556.773,A -85,B 0,C 180,E1 -26041.471,E2 -26041.471} C_VEL
LIN {X 0,Y 129.529,Z 554.693,A -85,B 0,C 180,E1 -26050.633,E2 -26050.633} C_VEL
LIN {X 0,Y 141.121,Z 551.536,A -85,B 0,C 180,E1 -26058.342,E2 -26058.342} C_VEL
LIN {X 0,Y 150.388,Z 548.964,A -85,B 0,C 180,E1 -26062.613,E2 -26062.613} C_VEL
LIN {X 0,Y 151.372,Z 548.278,A -85,B 0,C 180,E1 -26063.721,E2 -26063.721} C_VEL
LIN {X 0,Y 143.403,Z 546.474,A -85,B 0,C 180,E1 -26067.379,E2 -26067.379} C_VEL
LIN {X 0,Y 133.747,Z 542.677,A -85,B 0,C 180,E1 -26073.304,E2 -26073.304} C_VEL
LIN {X 0,Y 130.566,Z 540.832,A -85,B 0,C 180,E1 -26075.747,E2 -26075.747} C_VEL
LIN {X 0,Y 127.5,Z 539.122,A -85,B 0,C 180,E1 -26077.852,E2 -26077.852} C_VEL
LIN {X 0,Y 121.282,Z 535.98,A -85,B 0,C 180,E1 -26081.095,E2 -26081.095} C_VEL
LIN {X 0,Y 115.562,Z 532.26,A -85,B 0,C 180,E1 -26084.591,E2 -26084.591} C_VEL
LIN {X 0,Y 113.384,Z 529.706,A -85,B 0,C 180,E1 -26087.045,E2 -26087.045} C_VEL
LIN {X 0,Y 110.36,Z 522.668,A -85,B 0,C 180,E1 -26093.603,E2 -26093.603} C_VEL
LIN {X 0,Y 108.769,Z 513.655,A -85,B 0,C 180,E1 -26100.927,E2 -26100.927} C_VEL
LIN {X 0,Y 108.661,Z 504.247,A -85,B 0,C 180,E1 -26107.434,E2 -26107.434} C_VEL
LIN {X 0,Y 109.846,Z 492.861,A -85,B 0,C 180,E1 -26114.125,E2 -26114.125} C_VEL
LIN {X 0,Y 111.325,Z 483.202,A -85,B 0,C 180,E1 -26118.906,E2 -26118.906} C_VEL
LIN {X 0,Y 111.831,Z 483.264,A -85,B 0,C 180,E1 -26120.031,E2 -26120.031} C_VEL
LIN {X 0,Y 114.016,Z 481.902,A -85,B 0,C 180,E1 -26122.371,E2 -26122.371} C_VEL
LIN {X 0,Y 117.635,Z 478.691,A -85,B 0,C 180,E1 -26124.723,E2 -26124.723} C_VEL
LIN {X 0,Y 121.329,Z 476.459,A -85,B 0,C 180,E1 -26127.608,E2 -26127.608} C_VEL
LIN {X 0,Y 124.318,Z 474.145,A -85,B 0,C 180,E1 -26129.285,E2 -26129.285} C_VEL
LIN {X 0,Y 128.769,Z 470.112,A -85,B 0,C 180,E1 -26131.233,E2 -26131.233} C_VEL
LIN {X 0,Y 130.903,Z 468.932,A -85,B 0,C 180,E1 -26132.473,E2 -26132.473} C_VEL
LIN {X 0,Y 134.69,Z 466.037,A -85,B 0,C 180,E1 -26134.121,E2 -26134.121} C_VEL
LIN {X 0,Y 138.967,Z 461.904,A -85,B 0,C 180,E1 -26135.562,E2 -26135.562} C_VEL
LIN {X 0,Y 142.119,Z 458.337,A -85,B 0,C 180,E1 -26136.401,E2 -26136.401} C_VEL
LIN {X 0,Y 144.672,Z 456.425,A -85,B 0,C 180,E1 -26137.391,E2 -26137.391} C_VEL
LIN {X 0,Y 146.798,Z 456.005,A -85,B 0,C 180,E1 -26138.491,E2 -26138.491} C_VEL
LIN {X 0,Y 147.292,Z 464.941,A -85,B 0,C 180,E1 -26141.468,E2 -26141.468} C_VEL
LIN {X 0,Y 147.319,Z 467.545,A -85,B 0,C 180,E1 -26142.353,E2 -26142.353} C_VEL
LIN {X 0,Y 145.972,Z 471.733,A -85,B 0,C 180,E1 -26143.191,E2 -26143.191} C_VEL
LIN {X 0,Y 141.274,Z 483.256,A -85,B 0,C 180,E1 -26145.848,E2 -26145.848} C_VEL
LIN {X 0,Y 137.336,Z 491.454,A -85,B 0,C 180,E1 -26148.29,E2 -26148.29} C_VEL
LIN {X 0,Y 132.718,Z 499.938,A -85,B 0,C 180,E1 -26151.514,E2 -26151.514} C_VEL
LIN {X 0,Y 128.187,Z 507.196,A -85,B 0,C 180,E1 -26155.037,E2 -26155.037} C_VEL
LIN {X 0,Y 123.73,Z 513.768,A -85,B 0,C 180,E1 -26159.247,E2 -26159.247} C_VEL
LIN {X 0,Y 119.524,Z 519.214,A -85,B 0,C 180,E1 -26163.824,E2 -26163.824} C_VEL
LIN {X 0,Y 115.724,Z 523.523,A -85,B 0,C 180,E1 -26168.622,E2 -26168.622} C_VEL
LIN {X 0,Y 113.905,Z 525.741,A -85,B 0,C 180,E1 -26172.022,E2 -26172.022} C_VEL
LIN {X 0,Y 112.434,Z 527.543,A -85,B 0,C 180,E1 -26175.512,E2 -26175.512} C_VEL
LIN {X 0,Y 111.404,Z 528.894,A -85,B 0,C 180,E1 -26179.082,E2 -26179.082} C_VEL
LIN {X 0,Y 110.061,Z 530.449,A -85,B 0,C 180,E1 -26186.33,E2 -26186.33} C_VEL
LIN {X 0,Y 109.885,Z 530.673,A -85,B 0,C 180,E1 -26189.991,E2 -26189.991} C_VEL
LIN {X 0,Y 110.525,Z 529.908,A -85,B 0,C 180,E1 -26197.297,E2 -26197.297} C_VEL
LIN {X 0,Y 111.4,Z 528.958,A -85,B 0,C 180,E1 -26200.901,E2 -26200.901} C_VEL
LIN {X 0,Y 112.416,Z 527.647,A -85,B 0,C 180,E1 -26204.472,E2 -26204.472} C_VEL
LIN {X 0,Y 114.71,Z 524.853,A -85,B 0,C 180,E1 -26209.683,E2 -26209.683} C_VEL
LIN {X 0,Y 118.069,Z 520.985,A -85,B 0,C 180,E1 -26214.615,E2 -26214.615} C_VEL
LIN {X 0,Y 122.191,Z 515.955,A -85,B 0,C 180,E1 -26219.258,E2 -26219.258} C_VEL
LIN {X 0,Y 126.888,Z 509.409,A -85,B 0,C 180,E1 -26223.816,E2 -26223.816} C_VEL
LIN {X 0,Y 131.679,Z 501.822,A -85,B 0,C 180,E1 -26227.853,E2 -26227.853} C_VEL
LIN {X 0,Y 136.295,Z 493.773,A -85,B 0,C 180,E1 -26231.095,E2 -26231.095} C_VEL
LIN {X 0,Y 140.66,Z 484.953,A -85,B 0,C 180,E1 -26233.878,E2 -26233.878} C_VEL
LIN {X 0,Y 145.231,Z 473.973,A -85,B 0,C 180,E1 -26236.531,E2 -26236.531} C_VEL
LIN {X 0,Y 147.46,Z 467.803,A -85,B 0,C 180,E1 -26237.725,E2 -26237.725} C_VEL
LIN {X 0,Y 147.199,Z 459.154,A -85,B 0,C 180,E1 -26240.645,E2 -26240.645} C_VEL
LIN {X 0,Y 146.604,Z 453.849,A -85,B 0,C 180,E1 -26242.472,E2 -26242.472} C_VEL
LIN {X 0,Y 143.704,Z 445.364,A -85,B 0,C 180,E1 -26246.313,E2 -26246.313} C_VEL
LIN {X 0,Y 140.749,Z 438.83,A -85,B 0,C 180,E1 -26249.733,E2 -26249.733} C_VEL
LIN {X 0,Y 138.033,Z 434.117,A -85,B 0,C 180,E1 -26252.725,E2 -26252.725} C_VEL
LIN {X 0,Y 135.939,Z 430.584,A -85,B 0,C 180,E1 -26255.16,E2 -26255.16} C_VEL
LIN {X 0,Y 133.086,Z 426.626,A -85,B 0,C 180,E1 -26258.711,E2 -26258.711} C_VEL
LIN {X 0,Y 133.504,Z 423.876,A -85,B 0,C 180,E1 -26264.738,E2 -26264.738} C_VEL
LIN {X 0,Y 133.78,Z 422.683,A -85,B 0,C 180,E1 -26267.868,E2 -26267.868} C_VEL
LIN {X 0,Y 134.51,Z 421.439,A -85,B 0,C 180,E1 -26273.017,E2 -26273.017} C_VEL
LIN {X 0,Y 135.883,Z 420.675,A -85,B 0,C 180,E1 -26279.999,E2 -26279.999} C_VEL
LIN {X 0,Y 136.156,Z 421.377,A -85,B 0,C 180,E1 -26282.958,E2 -26282.958} C_VEL
LIN {X 0,Y 135.761,Z 424.872,A -85,B 0,C 180,E1 -26288.933,E2 -26288.933} C_VEL
LIN {X 0,Y 136.002,Z 429.604,A -85,B 0,C 180,E1 -26294.973,E2 -26294.973} C_VEL
LIN {X 0,Y 136.551,Z 436.026,A -85,B 0,C 180,E1 -26301.116,E2 -26301.116} C_VEL
LIN {X 0,Y 137.08,Z 441.483,A -85,B 0,C 180,E1 -26305.325,E2 -26305.325} C_VEL
LIN {X 0,Y 141.718,Z 451.625,A -85,B 0,C 180,E1 -26309.933,E2 -26309.933} C_VEL
LIN {X 0,Y 143.593,Z 458.2,A -85,B 0,C 180,E1 -26311.951,E2 -26311.951} C_VEL
LIN {X 0,Y 143.263,Z 470.364,A -85,B 0,C 180,E1 -26313.808,E2 -26313.808} C_VEL
LIN {X 0,Y 142.241,Z 483.867,A -85,B 0,C 180,E1 -26316.362,E2 -26316.362} C_VEL
LIN {X 0,Y 141.318,Z 487.682,A -85,B 0,C 180,E1 -26316.96,E2 -26316.96} C_VEL
LIN {X 0,Y 137.563,Z 499.091,A -85,B 0,C 180,E1 -26318.833,E2 -26318.833} C_VEL
LIN {X 0,Y 133.725,Z 508.85,A -85,B 0,C 180,E1 -26320.945,E2 -26320.945} C_VEL
LIN {X 0,Y 129.079,Z 519.125,A -85,B 0,C 180,E1 -26323.84,E2 -26323.84} C_VEL
LIN {X 0,Y 123.816,Z 529.425,A -85,B 0,C 180,E1 -26327.732,E2 -26327.732} C_VEL
LIN {X 0,Y 119.347,Z 537.575,A -85,B 0,C 180,E1 -26331.818,E2 -26331.818} C_VEL
LIN {X 0,Y 115.103,Z 544.957,A -85,B 0,C 180,E1 -26336.677,E2 -26336.677} C_VEL
LIN {X 0,Y 111.514,Z 551.528,A -85,B 0,C 180,E1 -26342.525,E2 -26342.525} C_VEL
LIN {X 0,Y 108.957,Z 557.01,A -85,B 0,C 180,E1 -26349.231,E2 -26349.231} C_VEL
LIN {X 0,Y 107.863,Z 560.299,A -85,B 0,C 180,E1 -26354.902,E2 -26354.902} C_VEL
LIN {X 0,Y 107.677,Z 561.93,A -85,B 0,C 180,E1 -26358.718,E2 -26358.718} C_VEL
LIN {X 0,Y 107.762,Z 563.116,A -85,B 0,C 180,E1 -26362.515,E2 -26362.515} C_VEL
LIN {X 0,Y 108.06,Z 563.873,A -85,B 0,C 180,E1 -26366.28,E2 -26366.28} C_VEL
LIN {X 0,Y 108.704,Z 564.219,A -85,B 0,C 180,E1 -26370.009,E2 -26370.009} C_VEL
LIN {X 0,Y 108.166,Z 563.874,A -85,B 0,C 180,E1 -26373.734,E2 -26373.734} C_VEL
LIN {X 0,Y 107.873,Z 563.107,A -85,B 0,C 180,E1 -26377.496,E2 -26377.496} C_VEL
LIN {X 0,Y 107.85,Z 561.566,A -85,B 0,C 180,E1 -26382.193,E2 -26382.193} C_VEL
LIN {X 0,Y 108.919,Z 558.196,A -85,B 0,C 180,E1 -26388.831,E2 -26388.831} C_VEL
LIN {X 0,Y 110.378,Z 555.467,A -85,B 0,C 180,E1 -26392.963,E2 -26392.963} C_VEL
LIN {X 0,Y 115.218,Z 554.796,A -85,B 0,C 180,E1 -26403.306,E2 -26403.306} C_VEL
LIN {X 0,Y 124.244,Z 552.97,A -85,B 0,C 180,E1 -26412.759,E2 -26412.759} C_VEL
LIN {X 0,Y 136.485,Z 550.203,A -85,B 0,C 180,E1 -26420.579,E2 -26420.579} C_VEL
LIN {X 0,Y 141.207,Z 549.071,A -85,B 0,C 180,E1 -26422.791,E2 -26422.791} C_VEL
LIN {X 0,Y 142.138,Z 548.613,A -85,B 0,C 180,E1 -26423.607,E2 -26423.607} C_VEL
LIN {X 0,Y 133.179,Z 545.778,A -85,B 0,C 180,E1 -26428.15,E2 -26428.15} C_VEL
LIN {X 0,Y 124.254,Z 541.199,A -85,B 0,C 180,E1 -26434.309,E2 -26434.309} C_VEL
LIN {X 0,Y 117.684,Z 535.66,A -85,B 0,C 180,E1 -26440.826,E2 -26440.826} C_VEL
LIN {X 0,Y 113.384,Z 529.706,A -85,B 0,C 180,E1 -26447.045,E2 -26447.045} C_VEL
LIN {X 0,Y 111.415,Z 527.044,A -85,B 0,C 180,E1 -26449.534,E2 -26449.534} C_VEL
LIN {X 0,Y 106.855,Z 522.265,A -85,B 0,C 180,E1 -26453.419,E2 -26453.419} C_VEL
LIN {X 0,Y 102.824,Z 516.97,A -85,B 0,C 180,E1 -26457.477,E2 -26457.477} C_VEL
LIN {X 0,Y 101.773,Z 513.556,A -85,B 0,C 180,E1 -26460.135,E2 -26460.135} C_VEL
LIN {X 0,Y 101.574,Z 504.277,A -85,B 0,C 180,E1 -26466.956,E2 -26466.956} C_VEL
LIN {X 0,Y 102.665,Z 493.29,A -85,B 0,C 180,E1 -26473.864,E2 -26473.864} C_VEL
LIN {X 0,Y 103.321,Z 493.085,A -85,B 0,C 180,E1 -26475.79,E2 -26475.79} C_VEL
LIN {X 0,Y 105.004,Z 491.862,A -85,B 0,C 180,E1 -26478.038,E2 -26478.038} C_VEL
LIN {X 0,Y 108.255,Z 489.139,A -85,B 0,C 180,E1 -26480.922,E2 -26480.922} C_VEL
LIN {X 0,Y 111.361,Z 487.414,A -85,B 0,C 180,E1 -26484.196,E2 -26484.196} C_VEL
LIN {X 0,Y 115.957,Z 483.878,A -85,B 0,C 180,E1 -26487.039,E2 -26487.039} C_VEL
LIN {X 0,Y 120,Z 481.584,A -85,B 0,C 180,E1 -26489.857,E2 -26489.857} C_VEL
LIN {X 0,Y 124.187,Z 478.522,A -85,B 0,C 180,E1 -26491.897,E2 -26491.897} C_VEL
LIN {X 0,Y 127.893,Z 475.498,A -85,B 0,C 180,E1 -26493.336,E2 -26493.336} C_VEL
LIN {X 0,Y 130.201,Z 474.227,A -85,B 0,C 180,E1 -26494.527,E2 -26494.527} C_VEL
LIN {X 0,Y 134.139,Z 471.428,A -85,B 0,C 180,E1 -26496.081,E2 -26496.081} C_VEL
LIN {X 0,Y 138.66,Z 467.54,A -85,B 0,C 180,E1 -26497.463,E2 -26497.463} C_VEL
LIN {X 0,Y 141.874,Z 464.379,A -85,B 0,C 180,E1 -26498.26,E2 -26498.26} C_VEL
LIN {X 0,Y 142.4,Z 465.549,A -85,B 0,C 180,E1 -26498.997,E2 -26498.997} C_VEL
LIN {X 0,Y 142.078,Z 470.687,A -85,B 0,C 180,E1 -26500.741,E2 -26500.741} C_VEL
LIN {X 0,Y 137.937,Z 480.842,A -85,B 0,C 180,E1 -26502.902,E2 -26502.902} C_VEL
LIN {X 0,Y 133.16,Z 490.654,A -85,B 0,C 180,E1 -26505.619,E2 -26505.619} C_VEL
LIN {X 0,Y 128.221,Z 499.451,A -85,B 0,C 180,E1 -26508.863,E2 -26508.863} C_VEL
LIN {X 0,Y 123.485,Z 506.835,A -85,B 0,C 180,E1 -26512.373,E2 -26512.373} C_VEL
LIN {X 0,Y 118.834,Z 513.413,A -85,B 0,C 180,E1 -26516.476,E2 -26516.476} C_VEL
LIN {X 0,Y 114.646,Z 518.605,A -85,B 0,C 180,E1 -26520.623,E2 -26520.623} C_VEL
LIN {X 0,Y 110.594,Z 523.259,A -85,B 0,C 180,E1 -26525.594,E2 -26525.594} C_VEL
LIN {X 0,Y 108.163,Z 525.787,A -85,B 0,C 180,E1 -26529.052,E2 -26529.052} C_VEL
LIN {X 0,Y 105.651,Z 528.621,A -85,B 0,C 180,E1 -26534.559,E2 -26534.559} C_VEL
LIN {X 0,Y 104.52,Z 529.972,A -85,B 0,C 180,E1 -26538.353,E2 -26538.353} C_VEL
LIN {X 0,Y 103.066,Z 531.525,A -85,B 0,C 180,E1 -26546.081,E2 -26546.081} C_VEL
LIN {X 0,Y 102.872,Z 531.749,A -85,B 0,C 180,E1 -26549.99,E2 -26549.99} C_VEL
LIN {X 0,Y 103.578,Z 530.983,A -85,B 0,C 180,E1 -26557.79,E2 -26557.79} C_VEL
LIN {X 0,Y 104.515,Z 530.035,A -85,B 0,C 180,E1 -26561.628,E2 -26561.628} C_VEL
LIN {X 0,Y 105.632,Z 528.723,A -85,B 0,C 180,E1 -26565.424,E2 -26565.424} C_VEL
LIN {X 0,Y 108.126,Z 525.928,A -85,B 0,C 180,E1 -26570.936,E2 -26570.936} C_VEL
LIN {X 0,Y 111.728,Z 522.06,A -85,B 0,C 180,E1 -26576.114,E2 -26576.114} C_VEL
LIN {X 0,Y 116.121,Z 517.027,A -85,B 0,C 180,E1 -26580.95,E2 -26580.95} C_VEL
LIN {X 0,Y 121.206,Z 510.37,A -85,B 0,C 180,E1 -26585.728,E2 -26585.728} C_VEL
LIN {X 0,Y 126.211,Z 502.892,A -85,B 0,C 180,E1 -26589.808,E2 -26589.808} C_VEL
LIN {X 0,Y 131.091,Z 494.839,A -85,B 0,C 180,E1 -26593.11,E2 -26593.11} C_VEL
LIN {X 0,Y 135.686,Z 486.016,A -85,B 0,C 180,E1 -26595.933,E2 -26595.933} C_VEL
LIN {X 0,Y 140.501,Z 475.029,A -85,B 0,C 180,E1 -26598.606,E2 -26598.606} C_VEL
LIN {X 0,Y 142.45,Z 469.759,A -85,B 0,C 180,E1 -26599.672,E2 -26599.672} C_VEL
LIN {X 0,Y 142.427,Z 461.025,A -85,B 0,C 180,E1 -26602.808,E2 -26602.808} C_VEL
LIN {X 0,Y 142.294,Z 458.72,A -85,B 0,C 180,E1 -26603.65,E2 -26603.65} C_VEL
LIN {X 0,Y 140.093,Z 450.803,A -85,B 0,C 180,E1 -26607.449,E2 -26607.449} C_VEL
LIN {X 0,Y 137.619,Z 444.482,A -85,B 0,C 180,E1 -26610.976,E2 -26610.976} C_VEL
LIN {X 0,Y 135.418,Z 440.093,A -85,B 0,C 180,E1 -26613.926,E2 -26613.926} C_VEL
LIN {X 0,Y 133.683,Z 436.786,A -85,B 0,C 180,E1 -26616.367,E2 -26616.367} C_VEL
LIN {X 0,Y 130.792,Z 432.486,A -85,B 0,C 180,E1 -26620.579,E2 -26620.579} C_VEL
LIN {X 0,Y 128.358,Z 428.56,A -85,B 0,C 180,E1 -26625.33,E2 -26625.33} C_VEL
LIN {X 0,Y 129.152,Z 427.045,A -85,B 0,C 180,E1 -26630.603,E2 -26630.603} C_VEL
LIN {X 0,Y 129.609,Z 426.396,A -85,B 0,C 180,E1 -26633.773,E2 -26633.773} C_VEL
LIN {X 0,Y 130.999,Z 425.875,A -85,B 0,C 180,E1 -26639.999,E2 -26639.999} C_VEL
LIN {X 0,Y 131.183,Z 426.708,A -85,B 0,C 180,E1 -26643.07,E2 -26643.07} C_VEL
LIN {X 0,Y 130.83,Z 430.462,A -85,B 0,C 180,E1 -26649.273,E2 -26649.273} C_VEL
LIN {X 0,Y 131.005,Z 434.232,A -85,B 0,C 180,E1 -26654.127,E2 -26654.127} C_VEL
LIN {X 0,Y 131.38,Z 439.582,A -85,B 0,C 180,E1 -26659.429,E2 -26659.429} C_VEL
LIN {X 0,Y 134.98,Z 448.146,A -85,B 0,C 180,E1 -26664.294,E2 -26664.294} C_VEL
LIN {X 0,Y 138.445,Z 456.539,A -85,B 0,C 180,E1 -26668.314,E2 -26668.314} C_VEL
LIN {X 0,Y 139.544,Z 461.681,A -85,B 0,C 180,E1 -26669.927,E2 -26669.927} C_VEL
LIN {X 0,Y 138.742,Z 473.741,A -85,B 0,C 180,E1 -26671.96,E2 -26671.96} C_VEL
LIN {X 0,Y 137.121,Z 486.612,A -85,B 0,C 180,E1 -26674.562,E2 -26674.562} C_VEL
LIN {X 0,Y 133.096,Z 498.173,A -85,B 0,C 180,E1 -26676.445,E2 -26676.445} C_VEL
LIN {X 0,Y 128.543,Z 509.019,A -85,B 0,C 180,E1 -26678.835,E2 -26678.835} C_VEL
LIN {X 0,Y 124.158,Z 518.022,A -85,B 0,C 180,E1 -26681.421,E2 -26681.421} C_VEL
LIN {X 0,Y 118.603,Z 528.209,A -85,B 0,C 180,E1 -26685.321,E2 -26685.321} C_VEL
LIN {X 0,Y 113.726,Z 536.467,A -85,B 0,C 180,E1 -26689.556,E2 -26689.556} C_VEL
LIN {X 0,Y 109.126,Z 543.85,A -85,B 0,C 180,E1 -26694.588,E2 -26694.588} C_VEL
LIN {X 0,Y 105.445,Z 549.821,A -85,B 0,C 180,E1 -26700.047,E2 -26700.047} C_VEL
LIN {X 0,Y 102.874,Z 554.549,A -85,B 0,C 180,E1 -26705.813,E2 -26705.813} C_VEL
LIN {X 0,Y 101.253,Z 558.194,A -85,B 0,C 180,E1 -26711.81,E2 -26711.81} C_VEL
LIN {X 0,Y 100.658,Z 560.831,A -85,B 0,C 180,E1 -26717.919,E2 -26717.919} C_VEL
LIN {X 0,Y 100.687,Z 562.02,A -85,B 0,C 180,E1 -26721.985,E2 -26721.985} C_VEL
LIN {X 0,Y 100.975,Z 562.784,A -85,B 0,C 180,E1 -26726.019,E2 -26726.019} C_VEL
LIN {X 0,Y 101.655,Z 563.137,A -85,B 0,C 180,E1 -26730.01,E2 -26730.01} C_VEL
LIN {X 0,Y 101.082,Z 562.784,A -85,B 0,C 180,E1 -26733.996,E2 -26733.996} C_VEL
LIN {X 0,Y 100.797,Z 562.01,A -85,B 0,C 180,E1 -26738.026,E2 -26738.026} C_VEL
LIN {X 0,Y 100.834,Z 560.627,A -85,B 0,C 180,E1 -26742.642,E2 -26742.642} C_VEL
LIN {X 0,Y 102.15,Z 557.094,A -85,B 0,C 180,E1 -26750.131,E2 -26750.131} C_VEL
LIN {X 0,Y 104.613,Z 553.135,A -85,B 0,C 180,E1 -26756.169,E2 -26756.169} C_VEL
LIN {X 0,Y 112.245,Z 552.237,A -85,B 0,C 180,E1 -26768.775,E2 -26768.775} C_VEL
LIN {X 0,Y 123.154,Z 550.398,A -85,B 0,C 180,E1 -26777.901,E2 -26777.901} C_VEL
LIN {X 0,Y 132.112,Z 548.673,A -85,B 0,C 180,E1 -26782.946,E2 -26782.946} C_VEL
LIN {X 0,Y 131.748,Z 548.039,A -85,B 0,C 180,E1 -26784.072,E2 -26784.072} C_VEL
LIN {X 0,Y 122.366,Z 544.015,A -85,B 0,C 180,E1 -26789.501,E2 -26789.501} C_VEL
LIN {X 0,Y 113.982,Z 538.364,A -85,B 0,C 180,E1 -26796.374,E2 -26796.374} C_VEL
LIN {X 0,Y 107.266,Z 530.596,A -85,B 0,C 180,E1 -26804.808,E2 -26804.808} C_VEL
LIN {X 0,Y 103.326,Z 521.855,A -85,B 0,C 180,E1 -26813.165,E2 -26813.165} C_VEL
LIN {X 0,Y 101.773,Z 513.556,A -85,B 0,C 180,E1 -26820.135,E2 -26820.135} C_VEL
LIN {X 0,Y 100.891,Z 511.211,A -85,B 0,C 180,E1 -26821.886,E2 -26821.886} C_VEL
LIN {X 0,Y 95.388,Z 504.016,A -85,B 0,C 180,E1 -26827.086,E2 -26827.086} C_VEL
LIN {X 0,Y 94.894,Z 502.369,A -85,B 0,C 180,E1 -26829.227,E2 -26829.227} C_VEL
LIN {X 0,Y 95.039,Z 502.116,A -85,B 0,C 180,E1 -26829.795,E2 -26829.795} C_VEL
LIN {X 0,Y 96.247,Z 501.06,A -85,B 0,C 180,E1 -26832.656,E2 -26832.656} C_VEL
LIN {X 0,Y 98.61,Z 499.009,A -85,B 0,C 180,E1 -26835.797,E2 -26835.797} C_VEL
LIN {X 0,Y 101.853,Z 496.889,A -85,B 0,C 180,E1 -26840.184,E2 -26840.184} C_VEL
LIN {X 0,Y 105.724,Z 494.185,A -85,B 0,C 180,E1 -26843.508,E2 -26843.508} C_VEL
LIN {X 0,Y 109.357,Z 492.181,A -85,B 0,C 180,E1 -26846.737,E2 -26846.737} C_VEL
LIN {X 0,Y 114.187,Z 488.852,A -85,B 0,C 180,E1 -26849.499,E2 -26849.499} C_VEL
LIN {X 0,Y 118.629,Z 486.489,A -85,B 0,C 180,E1 -26852.223,E2 -26852.223} C_VEL
LIN {X 0,Y 124.022,Z 482.789,A -85,B 0,C 180,E1 -26854.52,E2 -26854.52} C_VEL
LIN {X 0,Y 126.949,Z 480.651,A -85,B 0,C 180,E1 -26855.543,E2 -26855.543} C_VEL
LIN {X 0,Y 129.435,Z 479.331,A -85,B 0,C 180,E1 -26856.676,E2 -26856.676} C_VEL
LIN {X 0,Y 135.134,Z 475.439,A -85,B 0,C 180,E1 -26858.617,E2 -26858.617} C_VEL
LIN {X 0,Y 136.084,Z 475.421,A -85,B 0,C 180,E1 -26859.215,E2 -26859.215} C_VEL
LIN {X 0,Y 130.996,Z 486.528,A -85,B 0,C 180,E1 -26861.883,E2 -26861.883} C_VEL
LIN {X 0,Y 127.215,Z 493.595,A -85,B 0,C 180,E1 -26864.085,E2 -26864.085} C_VEL
LIN {X 0,Y 122.046,Z 502.085,A -85,B 0,C 180,E1 -26867.41,E2 -26867.41} C_VEL
LIN {X 0,Y 116.995,Z 509.339,A -85,B 0,C 180,E1 -26871.107,E2 -26871.107} C_VEL
LIN {X 0,Y 111.916,Z 515.917,A -85,B 0,C 180,E1 -26875.576,E2 -26875.576} C_VEL
LIN {X 0,Y 107.108,Z 521.367,A -85,B 0,C 180,E1 -26880.51,E2 -26880.51} C_VEL
LIN {X 0,Y 102.783,Z 525.677,A -85,B 0,C 180,E1 -26885.769,E2 -26885.769} C_VEL
LIN {X 0,Y 100.64,Z 527.897,A -85,B 0,C 180,E1 -26889.554,E2 -26889.554} C_VEL
LIN {X 0,Y 98.902,Z 529.699,A -85,B 0,C 180,E1 -26893.477,E2 -26893.477} C_VEL
LIN {X 0,Y 97.655,Z 531.05,A -85,B 0,C 180,E1 -26897.521,E2 -26897.521} C_VEL
LIN {X 0,Y 96.072,Z 532.601,A -85,B 0,C 180,E1 -26905.795,E2 -26905.795} C_VEL
LIN {X 0,Y 95.858,Z 532.825,A -85,B 0,C 180,E1 -26909.99,E2 -26909.99} C_VEL
LIN {X 0,Y 96.656,Z 532.056,A -85,B 0,C 180,E1 -26918.351,E2 -26918.351} C_VEL
LIN {X 0,Y 97.648,Z 531.112,A -85,B 0,C 180,E1 -26922.459,E2 -26922.459} C_VEL
LIN {X 0,Y 98.882,Z 529.8,A -85,B 0,C 180,E1 -26926.506,E2 -26926.506} C_VEL
LIN {X 0,Y 101.601,Z 527.004,A -85,B 0,C 180,E1 -26932.35,E2 -26932.35} C_VEL
LIN {X 0,Y 105.472,Z 523.134,A -85,B 0,C 180,E1 -26937.792,E2 -26937.792} C_VEL
LIN {X 0,Y 110.164,Z 518.1,A -85,B 0,C 180,E1 -26942.827,E2 -26942.827} C_VEL
LIN {X 0,Y 115.581,Z 511.435,A -85,B 0,C 180,E1 -26947.768,E2 -26947.768} C_VEL
LIN {X 0,Y 120.903,Z 503.962,A -85,B 0,C 180,E1 -26951.938,E2 -26951.938} C_VEL
LIN {X 0,Y 126.058,Z 495.905,A -85,B 0,C 180,E1 -26955.291,E2 -26955.291} C_VEL
LIN {X 0,Y 130.905,Z 487.077,A -85,B 0,C 180,E1 -26958.139,E2 -26958.139} C_VEL
LIN {X 0,Y 135.963,Z 476.086,A -85,B 0,C 180,E1 -26960.824,E2 -26960.824} C_VEL
LIN {X 0,Y 137.595,Z 471.801,A -85,B 0,C 180,E1 -26961.734,E2 -26961.734} C_VEL
LIN {X 0,Y 137.888,Z 464.228,A -85,B 0,C 180,E1 -26964.623,E2 -26964.623} C_VEL
LIN {X 0,Y 137.295,Z 459.946,A -85,B 0,C 180,E1 -26966.612,E2 -26966.612} C_VEL
LIN {X 0,Y 135.759,Z 454.168,A -85,B 0,C 180,E1 -26969.746,E2 -26969.746} C_VEL
LIN {X 0,Y 133.944,Z 449.063,A -85,B 0,C 180,E1 -26972.943,E2 -26972.943} C_VEL
LIN {X 0,Y 132.318,Z 445.256,A -85,B 0,C 180,E1 -26975.691,E2 -26975.691} C_VEL
LIN {X 0,Y 131.136,Z 442.738,A -85,B 0,C 180,E1 -26977.758,E2 -26977.758} C_VEL
LIN {X 0,Y 129.025,Z 439.027,A -85,B 0,C 180,E1 -26981.541,E2 -26981.541} C_VEL
LIN {X 0,Y 126.798,Z 435.224,A -85,B 0,C 180,E1 -26986.374,E2 -26986.374} C_VEL
LIN {X 0,Y 124.707,Z 431.394,A -85,B 0,C 180,E1 -26994.339,E2 -26994.339} C_VEL
LIN {X 0,Y 126.088,Z 431.031,A -85,B 0,C 180,E1 -26999.999,E2 -26999.999} C_VEL
LIN {X 0,Y 126.198,Z 432.074,A -85,B 0,C 180,E1 -27003.191,E2 -27003.191} C_VEL
LIN {X 0,Y 125.869,Z 436.036,A -85,B 0,C 180,E1 -27009.642,E2 -27009.642} C_VEL
LIN {X 0,Y 127.926,Z 442.198,A -85,B 0,C 180,E1 -27015.258,E2 -27015.258} C_VEL
LIN {X 0,Y 129.57,Z 446.085,A -85,B 0,C 180,E1 -27018.274,E2 -27018.274} C_VEL
LIN {X 0,Y 132.282,Z 453.502,A -85,B 0,C 180,E1 -27022.654,E2 -27022.654} C_VEL
LIN {X 0,Y 135.169,Z 461.829,A -85,B 0,C 180,E1 -27026.851,E2 -27026.851} C_VEL
LIN {X 0,Y 135.563,Z 464.92,A -85,B 0,C 180,E1 -27027.812,E2 -27027.812} C_VEL
LIN {X 0,Y 134.246,Z 477.32,A -85,B 0,C 180,E1 -27030.1,E2 -27030.1} C_VEL
LIN {X 0,Y 132.405,Z 487.876,A -85,B 0,C 180,E1 -27032.332,E2 -27032.332} C_VEL
LIN {X 0,Y 127.777,Z 499.89,A -85,B 0,C 180,E1 -27034.424,E2 -27034.424} C_VEL
LIN {X 0,Y 123.55,Z 509.116,A -85,B 0,C 180,E1 -27036.551,E2 -27036.551} C_VEL
LIN {X 0,Y 118.367,Z 518.911,A -85,B 0,C 180,E1 -27039.492,E2 -27039.492} C_VEL
LIN {X 0,Y 113.007,Z 528.024,A -85,B 0,C 180,E1 -27043.163,E2 -27043.163} C_VEL
LIN {X 0,Y 107.399,Z 536.693,A -85,B 0,C 180,E1 -27047.889,E2 -27047.889} C_VEL
LIN {X 0,Y 102.532,Z 543.8,A -85,B 0,C 180,E1 -27053.16,E2 -27053.16} C_VEL
LIN {X 0,Y 98.129,Z 550.416,A -85,B 0,C 180,E1 -27059.924,E2 -27059.924} C_VEL
LIN {X 0,Y 95.541,Z 554.789,A -85,B 0,C 180,E1 -27066.147,E2 -27066.147} C_VEL
LIN {X 0,Y 94.004,Z 558.086,A -85,B 0,C 180,E1 -27072.611,E2 -27072.611} C_VEL
LIN {X 0,Y 93.632,Z 559.838,A -85,B 0,C 180,E1 -27077.356,E2 -27077.356} C_VEL
LIN {X 0,Y 93.623,Z 560.925,A -85,B 0,C 180,E1 -27081.376,E2 -27081.376} C_VEL
LIN {X 0,Y 93.887,Z 561.694,A -85,B 0,C 180,E1 -27085.718,E2 -27085.718} C_VEL
LIN {X 0,Y 94.576,Z 562.05,A -85,B 0,C 180,E1 -27090.01,E2 -27090.01} C_VEL
LIN {X 0,Y 93.994,Z 561.693,A -85,B 0,C 180,E1 -27094.298,E2 -27094.298} C_VEL
LIN {X 0,Y 93.733,Z 560.915,A -85,B 0,C 180,E1 -27098.635,E2 -27098.635} C_VEL
LIN {X 0,Y 93.806,Z 559.682,A -85,B 0,C 180,E1 -27103.11,E2 -27103.11} C_VEL
LIN {X 0,Y 94.822,Z 557.09,A -85,B 0,C 180,E1 -27109.494,E2 -27109.494} C_VEL
LIN {X 0,Y 97.062,Z 553.479,A -85,B 0,C 180,E1 -27115.76,E2 -27115.76} C_VEL
LIN {X 0,Y 99.219,Z 550.625,A -85,B 0,C 180,E1 -27119.735,E2 -27119.735} C_VEL
LIN {X 0,Y 106.901,Z 550.054,A -85,B 0,C 180,E1 -27131.115,E2 -27131.115} C_VEL
LIN {X 0,Y 118.553,Z 548.451,A -85,B 0,C 180,E1 -27140.424,E2 -27140.424} C_VEL
LIN {X 0,Y 123.132,Z 547.766,A -85,B 0,C 180,E1 -27143.054,E2 -27143.054} C_VEL
LIN {X 0,Y 121.373,Z 546.666,A -85,B 0,C 180,E1 -27144.618,E2 -27144.618} C_VEL
LIN {X 0,Y 111.02,Z 540.895,A -85,B 0,C 180,E1 -27151.657,E2 -27151.657} C_VEL
LIN {X 0,Y 104.409,Z 535.108,A -85,B 0,C 180,E1 -27158.273,E2 -27158.273} C_VEL
LIN {X 0,Y 99.387,Z 528.137,A -85,B 0,C 180,E1 -27165.672,E2 -27165.672} C_VEL
LIN {X 0,Y 96.015,Z 519.763,A -85,B 0,C 180,E1 -27173.698,E2 -27173.698} C_VEL
LIN {X 0,Y 94.642,Z 511.179,A -85,B 0,C 180,E1 -27181.065,E2 -27181.065} C_VEL
LIN {X 0,Y 94.568,Z 502.579,A -85,B 0,C 180,E1 -27187.743,E2 -27187.743} C_VEL
LIN {X 0,Y 94.595,Z 502.569,A -85,B 0,C 180,E1 -27188.547,E2 -27188.547} C_VEL
LIN {X 0,Y 95.039,Z 502.116,A -85,B 0,C 180,E1 -27189.795,E2 -27189.795} C_VEL
LIN {X 0,Y 96.614,Z 500.995,A -85,B 0,C 180,E1 -27194.351,E2 -27194.351} C_VEL
LIN {X 0,Y 100.617,Z 499.852,A -85,B 0,C 180,E1 -27203.187,E2 -27203.187} C_VEL
LIN {X 0,Y 104.061,Z 498.455,A -85,B 0,C 180,E1 -27207.037,E2 -27207.037} C_VEL
LIN {X 0,Y 107.205,Z 496.803,A -85,B 0,C 180,E1 -27209.341,E2 -27209.341} C_VEL
LIN {X 0,Y 112.406,Z 493.594,A -85,B 0,C 180,E1 -27212.105,E2 -27212.105} C_VEL
LIN {X 0,Y 117.226,Z 491.161,A -85,B 0,C 180,E1 -27214.721,E2 -27214.721} C_VEL
LIN {X 0,Y 123.171,Z 487.414,A -85,B 0,C 180,E1 -27216.971,E2 -27216.971} C_VEL
LIN {X 0,Y 125.958,Z 485.565,A -85,B 0,C 180,E1 -27217.863,E2 -27217.863} C_VEL
LIN {X 0,Y 127.398,Z 484.859,A -85,B 0,C 180,E1 -27218.462,E2 -27218.462} C_VEL
LIN {X 0,Y 127.013,Z 486.465,A -85,B 0,C 180,E1 -27219.215,E2 -27219.215} C_VEL
LIN {X 0,Y 122.435,Z 494.667,A -85,B 0,C 180,E1 -27221.725,E2 -27221.725} C_VEL
LIN {X 0,Y 116.977,Z 503.159,A -85,B 0,C 180,E1 -27225.084,E2 -27225.084} C_VEL
LIN {X 0,Y 111.621,Z 510.414,A -85,B 0,C 180,E1 -27228.845,E2 -27228.845} C_VEL
LIN {X 0,Y 106.209,Z 516.992,A -85,B 0,C 180,E1 -27233.438,E2 -27233.438} C_VEL
LIN {X 0,Y 101.058,Z 522.444,A -85,B 0,C 180,E1 -27238.551,E2 -27238.551} C_VEL
LIN {X 0,Y 96.427,Z 526.754,A -85,B 0,C 180,E1 -27244.057,E2 -27244.057} C_VEL
LIN {X 0,Y 94.093,Z 528.975,A -85,B 0,C 180,E1 -27248.06,E2 -27248.06} C_VEL
LIN {X 0,Y 92.193,Z 530.777,A -85,B 0,C 180,E1 -27252.236,E2 -27252.236} C_VEL
LIN {X 0,Y 90.812,Z 532.127,A -85,B 0,C 180,E1 -27256.564,E2 -27256.564} C_VEL
LIN {X 0,Y 89.079,Z 533.677,A -85,B 0,C 180,E1 -27265.464,E2 -27265.464} C_VEL
LIN {X 0,Y 88.842,Z 533.902,A -85,B 0,C 180,E1 -27269.989,E2 -27269.989} C_VEL
LIN {X 0,Y 89.74,Z 533.129,A -85,B 0,C 180,E1 -27279,E2 -27279} C_VEL
LIN {X 0,Y 90.804,Z 532.189,A -85,B 0,C 180,E1 -27283.415,E2 -27283.415} C_VEL
LIN {X 0,Y 92.171,Z 530.876,A -85,B 0,C 180,E1 -27287.746,E2 -27287.746} C_VEL
LIN {X 0,Y 95.147,Z 528.079,A -85,B 0,C 180,E1 -27293.958,E2 -27293.958} C_VEL
LIN {X 0,Y 99.318,Z 524.208,A -85,B 0,C 180,E1 -27299.68,E2 -27299.68} C_VEL
LIN {X 0,Y 104.338,Z 519.172,A -85,B 0,C 180,E1 -27304.915,E2 -27304.915} C_VEL
LIN {X 0,Y 110.227,Z 512.381,A -85,B 0,C 180,E1 -27310.081,E2 -27310.081} C_VEL
LIN {X 0,Y 115.777,Z 505.031,A -85,B 0,C 180,E1 -27314.26,E2 -27314.26} C_VEL
LIN {X 0,Y 121.228,Z 496.971,A -85,B 0,C 180,E1 -27317.646,E2 -27317.646} C_VEL
LIN {X 0,Y 126.334,Z 488.139,A -85,B 0,C 180,E1 -27320.509,E2 -27320.509} C_VEL
LIN {X 0,Y 131.641,Z 477.143,A -85,B 0,C 180,E1 -27323.194,E2 -27323.194} C_VEL
LIN {X 0,Y 132.805,Z 474.554,A -85,B 0,C 180,E1 -27323.698,E2 -27323.698} C_VEL
LIN {X 0,Y 133.396,Z 467.754,A -85,B 0,C 180,E1 -27326.414,E2 -27326.414} C_VEL
LIN {X 0,Y 132.804,Z 462.979,A -85,B 0,C 180,E1 -27328.936,E2 -27328.936} C_VEL
LIN {X 0,Y 131.387,Z 456.689,A -85,B 0,C 180,E1 -27332.756,E2 -27332.756} C_VEL
LIN {X 0,Y 129.426,Z 450.992,A -85,B 0,C 180,E1 -27337.026,E2 -27337.026} C_VEL
LIN {X 0,Y 128.529,Z 448.787,A -85,B 0,C 180,E1 -27339.012,E2 -27339.012} C_VEL
LIN {X 0,Y 126.997,Z 445.512,A -85,B 0,C 180,E1 -27342.486,E2 -27342.486} C_VEL
LIN {X 0,Y 125.209,Z 441.829,A -85,B 0,C 180,E1 -27347.436,E2 -27347.436} C_VEL
LIN {X 0,Y 123.609,Z 438.321,A -85,B 0,C 180,E1 -27355.106,E2 -27355.106} C_VEL
LIN {X 0,Y 123.424,Z 437.818,A -85,B 0,C 180,E1 -27360.407,E2 -27360.407} C_VEL
LIN {X 0,Y 123.594,Z 439.1,A -85,B 0,C 180,E1 -27363.462,E2 -27363.462} C_VEL
LIN {X 0,Y 124.685,Z 443.296,A -85,B 0,C 180,E1 -27369.325,E2 -27369.325} C_VEL
LIN {X 0,Y 127.275,Z 451.417,A -85,B 0,C 180,E1 -27376.438,E2 -27376.438} C_VEL
LIN {X 0,Y 129.498,Z 459.139,A -85,B 0,C 180,E1 -27381.175,E2 -27381.175} C_VEL
LIN {X 0,Y 131.595,Z 466.421,A -85,B 0,C 180,E1 -27385.092,E2 -27385.092} C_VEL
LIN {X 0,Y 131.562,Z 468.486,A -85,B 0,C 180,E1 -27385.638,E2 -27385.638} C_VEL
LIN {X 0,Y 129.507,Z 481.843,A -85,B 0,C 180,E1 -27388.348,E2 -27388.348} C_VEL
LIN {X 0,Y 128.155,Z 488.144,A -85,B 0,C 180,E1 -27389.799,E2 -27389.799} C_VEL
LIN {X 0,Y 123.193,Z 500.238,A -85,B 0,C 180,E1 -27391.958,E2 -27391.958} C_VEL
LIN {X 0,Y 118.092,Z 510.385,A -85,B 0,C 180,E1 -27394.353,E2 -27394.353} C_VEL
LIN {X 0,Y 112.733,Z 519.782,A -85,B 0,C 180,E1 -27397.374,E2 -27397.374} C_VEL
LIN {X 0,Y 106.79,Z 528.909,A -85,B 0,C 180,E1 -27401.319,E2 -27401.319} C_VEL
LIN {X 0,Y 101.175,Z 536.864,A -85,B 0,C 180,E1 -27406.016,E2 -27406.016} C_VEL
LIN {X 0,Y 96.032,Z 543.753,A -85,B 0,C 180,E1 -27411.547,E2 -27411.547} C_VEL
LIN {X 0,Y 91.888,Z 549.299,A -85,B 0,C 180,E1 -27417.643,E2 -27417.643} C_VEL
LIN {X 0,Y 88.942,Z 553.675,A -85,B 0,C 180,E1 -27424.253,E2 -27424.253} C_VEL
LIN {X 0,Y 87.13,Z 556.978,A -85,B 0,C 180,E1 -27431.189,E2 -27431.189} C_VEL
LIN {X 0,Y 86.591,Z 558.896,A -85,B 0,C 180,E1 -27436.888,E2 -27436.888} C_VEL
LIN {X 0,Y 86.57,Z 559.83,A -85,B 0,C 180,E1 -27440.667,E2 -27440.667} C_VEL
LIN {X 0,Y 86.796,Z 560.602,A -85,B 0,C 180,E1 -27445.367,E2 -27445.367} C_VEL
LIN {X 0,Y 87.496,Z 560.964,A -85,B 0,C 180,E1 -27450.011,E2 -27450.011} C_VEL
LIN {X 0,Y 86.903,Z 560.602,A -85,B 0,C 180,E1 -27454.65,E2 -27454.65} C_VEL
LIN {X 0,Y 86.682,Z 559.819,A -85,B 0,C 180,E1 -27459.343,E2 -27459.343} C_VEL
LIN {X 0,Y 86.837,Z 558.616,A -85,B 0,C 180,E1 -27464.063,E2 -27464.063} C_VEL
LIN {X 0,Y 88.083,Z 555.988,A -85,B 0,C 180,E1 -27471.053,E2 -27471.053} C_VEL
LIN {X 0,Y 90.632,Z 552.374,A -85,B 0,C 180,E1 -27477.739,E2 -27477.739} C_VEL
LIN {X 0,Y 94.294,Z 548.054,A -85,B 0,C 180,E1 -27483.728,E2 -27483.728} C_VEL
LIN {X 0,Y 105.563,Z 547.317,A -85,B 0,C 180,E1 -27497.095,E2 -27497.095} C_VEL
LIN {X 0,Y 114.239,Z 546.347,A -85,B 0,C 180,E1 -27503.12,E2 -27503.12} C_VEL
LIN {X 0,Y 108.913,Z 543.367,A -85,B 0,C 180,E1 -27506.738,E2 -27506.738} C_VEL
LIN {X 0,Y 101.142,Z 537.8,A -85,B 0,C 180,E1 -27513.151,E2 -27513.151} C_VEL
LIN {X 0,Y 94.964,Z 531.117,A -85,B 0,C 180,E1 -27520.549,E2 -27520.549} C_VEL
LIN {X 0,Y 90.039,Z 522.069,A -85,B 0,C 180,E1 -27529.887,E2 -27529.887} C_VEL
LIN {X 0,Y 87.81,Z 512.374,A -85,B 0,C 180,E1 -27538.855,E2 -27538.855} C_VEL
LIN {X 0,Y 87.638,Z 510.971,A -85,B 0,C 180,E1 -27540.289,E2 -27540.289} C_VEL
LIN {X 0,Y 87.545,Z 510.664,A -85,B 0,C 180,E1 -27542.302,E2 -27542.302} C_VEL
LIN {X 0,Y 87.897,Z 509.985,A -85,B 0,C 180,E1 -27544.588,E2 -27544.588} C_VEL
LIN {X 0,Y 89.853,Z 507.777,A -85,B 0,C 180,E1 -27549.002,E2 -27549.002} C_VEL
LIN {X 0,Y 91.505,Z 506.406,A -85,B 0,C 180,E1 -27553.323,E2 -27553.323} C_VEL
LIN {X 0,Y 94.419,Z 504.182,A -85,B 0,C 180,E1 -27557.323,E2 -27557.323} C_VEL
LIN {X 0,Y 99.391,Z 501.143,A -85,B 0,C 180,E1 -27563.162,E2 -27563.162} C_VEL
LIN {X 0,Y 103.184,Z 498.888,A -85,B 0,C 180,E1 -27566.28,E2 -27566.28} C_VEL
LIN {X 0,Y 104.061,Z 498.455,A -85,B 0,C 180,E1 -27567.037,E2 -27567.037} C_VEL
LIN {X 0,Y 106.541,Z 497.691,A -85,B 0,C 180,E1 -27569.59,E2 -27569.59} C_VEL
LIN {X 0,Y 111.921,Z 497.251,A -85,B 0,C 180,E1 -27575.276,E2 -27575.276} C_VEL
LIN {X 0,Y 114.44,Z 496.301,A -85,B 0,C 180,E1 -27576.743,E2 -27576.743} C_VEL
LIN {X 0,Y 118.434,Z 494.202,A -85,B 0,C 180,E1 -27578.311,E2 -27578.311} C_VEL
LIN {X 0,Y 117.879,Z 495.739,A -85,B 0,C 180,E1 -27579.177,E2 -27579.177} C_VEL
LIN {X 0,Y 112.116,Z 504.233,A -85,B 0,C 180,E1 -27582.55,E2 -27582.55} C_VEL
LIN {X 0,Y 106.657,Z 511.229,A -85,B 0,C 180,E1 -27586.212,E2 -27586.212} C_VEL
LIN {X 0,Y 100.666,Z 518.067,A -85,B 0,C 180,E1 -27591.061,E2 -27591.061} C_VEL
LIN {X 0,Y 95.141,Z 523.521,A -85,B 0,C 180,E1 -27596.345,E2 -27596.345} C_VEL
LIN {X 0,Y 90.169,Z 527.831,A -85,B 0,C 180,E1 -27602.106,E2 -27602.106} C_VEL
LIN {X 0,Y 87.619,Z 530.053,A -85,B 0,C 180,E1 -27606.344,E2 -27606.344} C_VEL
LIN {X 0,Y 85.533,Z 531.854,A -85,B 0,C 180,E1 -27610.8,E2 -27610.8} C_VEL
LIN {X 0,Y 83.998,Z 533.205,A -85,B 0,C 180,E1 -27615.451,E2 -27615.451} C_VEL
LIN {X 0,Y 82.089,Z 534.754,A -85,B 0,C 180,E1 -27625.077,E2 -27625.077} C_VEL
LIN {X 0,Y 81.825,Z 534.979,A -85,B 0,C 180,E1 -27629.988,E2 -27629.988} C_VEL
